KUKA KRL program: EPS_2_25252_SD4A_A_20250910061723.src

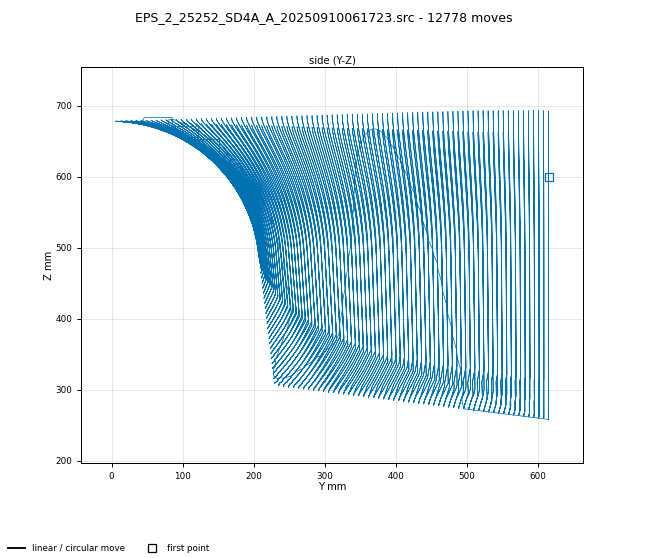
[picture p0: tool path of EPS_2_25252_SD4A_A_20250910061723.src, 12778 of 12780 moves have a stored position in this frame; points joined in program order, loops and branches not executed]
&ACCESS RVP
&REL 4
&COMMENT QRS 19112012
&PARAM EDITMASK = *
DEF PART()
EXT BAS (BAS_COMMAND :IN,REAL :IN )
INT I
BAS (#INITMOV,0 )

;KUKA QRS Post kuka4.cps  Date:22-06-2017 !

File_ID=2837

QRS_PRE_INIT()

;Init var - Until changes are made in qrs_pre_init
Outlet_Square_prg=0
Inlet_1_Square_prg=0
Inlet_2_Square_prg=0
Inlet_3_Square_prg=0
Inlet_4_Square_prg=0
Inlet_5_Square_prg=0

Outlet_1={X 0.000, Y 512.630, Z 510.000, B 0.000, E1 0.000 }
Inlet_1={X 0.000, Y 514.870, Z 480.000, B 0.000, E1 180.000 }
Outlet_1_type=366
Inlet_1_type=366
;QRS#1=Sidecore dimensions
;QRS#2=375-15" PVC SDR 35
;QRS#3=375-15" PVC SDR 35
;QRS#4=
;QRS#5=
;QRS#6=
;QRS#7=
;QRS#8=
;QRS#9=20Y PSX
;QRS#10=20Y PSX
;QRS#11=
;QRS#12=
;QRS#13=
;QRS#14=
;QRS#15=
;QRS#16=1220x127x991 3,25'
;QRS#17=EPS Height
;QRS#18=693
;QRS#19=*
;QRS#20= UPDATED VERSION 22-06-2017
;QRS#21=*
Outlet_Square=0250
Inlet_1_Square=0250
Inlet_2_Square=0
Inlet_3_Square=0
Inlet_4_Square=0
Inlet_5_Square=0
Mill_Square=1
Outlet_Square_Prg=252
Inlet_1_Square_prg=252

QRS_INIT()

$ADVANCE=5

; T1
PTP {E1 173.613,E2 173.613}
PTP {X 0,Y 615.489,A -85,B 0,C 180,E1 173.613,E2 173.613,E3 0,E4 0,E5 0,E6 0}
QRS_SPEED_INIT()
LIN {X 0,Y 615.489,Z 600,A -85,B 0,C 180,E1 173.613,E2 173.613,E3 0,E4 0,E5 0,E6 0} C_VEL
LIN {X 0,Y 615.489,Z 268.179,A -85,B 0,C 180,E1 173.613,E2 173.613} C_VEL
LIN {X 0,Y 615.489,Z 260.004,A -85,B 0,C 180,E1 173.613,E2 173.613} C_VEL
LIN {X 0,Y 615.477,Z 258.004,A -85,B 0,C 180,E1 173.427,E2 173.427} C_VEL
LIN {X 0,Y 615.484,Z 258.009,A -85,B 0,C 180,E1 170.801,E2 170.801} C_VEL
LIN {X 0,Y 615.489,Z 257.994,A -85,B 0,C 180,E1 168.139,E2 168.139} C_VEL
LIN {X 0,Y 615.478,Z 258.004,A -85,B 0,C 180,E1 165.451,E2 165.451} C_VEL
LIN {X 0,Y 615.479,Z 258.006,A -85,B 0,C 180,E1 162.729,E2 162.729} C_VEL
LIN {X 0,Y 615.488,Z 257.994,A -85,B 0,C 180,E1 159.967,E2 159.967} C_VEL
LIN {X 0,Y 615.485,Z 258.012,A -85,B 0,C 180,E1 157.155,E2 157.155} C_VEL
LIN {X 0,Y 615.476,Z 257.998,A -85,B 0,C 180,E1 154.284,E2 154.284} C_VEL
LIN {X 0,Y 615.481,Z 258.002,A -85,B 0,C 180,E1 151.55,E2 151.55} C_VEL
LIN {X 0,Y 615.478,Z 258.01,A -85,B 0,C 180,E1 148.915,E2 148.915} C_VEL
LIN {X 0,Y 615.493,Z 257.994,A -85,B 0,C 180,E1 145.978,E2 145.978} C_VEL
LIN {X 0,Y 615.483,Z 258.014,A -85,B 0,C 180,E1 143.063,E2 143.063} C_VEL
LIN {X 0,Y 615.476,Z 257.997,A -85,B 0,C 180,E1 140.249,E2 140.249} C_VEL
LIN {X 0,Y 615.484,Z 258.001,A -85,B 0,C 180,E1 137.647,E2 137.647} C_VEL
LIN {X 0,Y 615.479,Z 258.008,A -85,B 0,C 180,E1 134.931,E2 134.931} C_VEL
LIN {X 0,Y 615.488,Z 257.994,A -85,B 0,C 180,E1 132.08,E2 132.08} C_VEL
LIN {X 0,Y 615.486,Z 258.01,A -85,B 0,C 180,E1 129.062,E2 129.062} C_VEL
LIN {X 0,Y 615.469,Z 258,A -85,B 0,C 180,E1 126.426,E2 126.426} C_VEL
LIN {X 0,Y 615.487,Z 258.005,A -85,B 0,C 180,E1 123.534,E2 123.534} C_VEL
LIN {X 0,Y 615.47,Z 258.008,A -85,B 0,C 180,E1 120.92,E2 120.92} C_VEL
LIN {X 0,Y 615.467,Z 258,A -85,B 0,C 180,E1 118.447,E2 118.447} C_VEL
LIN {X 0,Y 615.488,Z 258.005,A -85,B 0,C 180,E1 115.569,E2 115.569} C_VEL
LIN {X 0,Y 615.477,Z 258.065,A -85,B 0,C 180,E1 114.239,E2 114.239} C_VEL
LIN {X 0,Y 615.49,Z 282.739,A -85,B 0,C 180,E1 111.982,E2 111.982} C_VEL
LIN {X 0,Y 615.49,Z 489.333,A -85,B 0,C 180,E1 109.424,E2 109.424} C_VEL
LIN {X 0,Y 615.49,Z 505.929,A -85,B 0,C 180,E1 109.078,E2 109.078} C_VEL
LIN {X 0,Y 615.495,Z 522.043,A -85,B 0,C 180,E1 108.607,E2 108.607} C_VEL
LIN {X 0,Y 615.494,Z 537.183,A -85,B 0,C 180,E1 108.038,E2 108.038} C_VEL
LIN {X 0,Y 615.496,Z 551.837,A -85,B 0,C 180,E1 107.356,E2 107.356} C_VEL
LIN {X 0,Y 615.497,Z 566.761,A -85,B 0,C 180,E1 106.51,E2 106.51} C_VEL
LIN {X 0,Y 615.496,Z 580.745,A -85,B 0,C 180,E1 105.565,E2 105.565} C_VEL
LIN {X 0,Y 615.497,Z 593.514,A -85,B 0,C 180,E1 104.549,E2 104.549} C_VEL
LIN {X 0,Y 615.498,Z 604.488,A -85,B 0,C 180,E1 103.537,E2 103.537} C_VEL
LIN {X 0,Y 615.488,Z 615.378,A -85,B 0,C 180,E1 102.363,E2 102.363} C_VEL
LIN {X 0,Y 615.487,Z 625.791,A -85,B 0,C 180,E1 101.041,E2 101.041} C_VEL
LIN {X 0,Y 615.495,Z 634.704,A -85,B 0,C 180,E1 99.696,E2 99.696} C_VEL
LIN {X 0,Y 615.488,Z 641.269,A -85,B 0,C 180,E1 98.537,E2 98.537} C_VEL
LIN {X 0,Y 615.494,Z 648.799,A -85,B 0,C 180,E1 96.897,E2 96.897} C_VEL
LIN {X 0,Y 615.495,Z 654.596,A -85,B 0,C 180,E1 95.241,E2 95.241} C_VEL
LIN {X 0,Y 615.496,Z 657.978,A -85,B 0,C 180,E1 93.928,E2 93.928} C_VEL
LIN {X 0,Y 615.486,Z 660.43,A -85,B 0,C 180,E1 92.618,E2 92.618} C_VEL
LIN {X 0,Y 615.489,Z 661.838,A -85,B 0,C 180,E1 91.309,E2 91.309} C_VEL
LIN {X 0,Y 615.491,Z 662.385,A -85,B 0,C 180,E1 90,E2 90} C_VEL
LIN {X 0,Y 615.486,Z 661.902,A -85,B 0,C 180,E1 88.691,E2 88.691} C_VEL
LIN {X 0,Y 615.486,Z 660.57,A -85,B 0,C 180,E1 87.382,E2 87.382} C_VEL
LIN {X 0,Y 615.493,Z 658.174,A -85,B 0,C 180,E1 86.072,E2 86.072} C_VEL
LIN {X 0,Y 615.49,Z 654.879,A -85,B 0,C 180,E1 84.759,E2 84.759} C_VEL
LIN {X 0,Y 615.491,Z 649.16,A -85,B 0,C 180,E1 83.103,E2 83.103} C_VEL
LIN {X 0,Y 615.497,Z 643.327,A -85,B 0,C 180,E1 81.794,E2 81.794} C_VEL
LIN {X 0,Y 615.492,Z 635.251,A -85,B 0,C 180,E1 80.304,E2 80.304} C_VEL
LIN {X 0,Y 615.493,Z 626.455,A -85,B 0,C 180,E1 78.959,E2 78.959} C_VEL
LIN {X 0,Y 615.491,Z 616.172,A -85,B 0,C 180,E1 77.638,E2 77.638} C_VEL
LIN {X 0,Y 615.495,Z 605.357,A -85,B 0,C 180,E1 76.463,E2 76.463} C_VEL
LIN {X 0,Y 615.495,Z 594.546,A -85,B 0,C 180,E1 75.451,E2 75.451} C_VEL
LIN {X 0,Y 615.497,Z 580.815,A -85,B 0,C 180,E1 74.35,E2 74.35} C_VEL
LIN {X 0,Y 615.498,Z 566.994,A -85,B 0,C 180,E1 73.414,E2 73.414} C_VEL
LIN {X 0,Y 615.492,Z 551.926,A -85,B 0,C 180,E1 72.558,E2 72.558} C_VEL
LIN {X 0,Y 615.487,Z 535.522,A -85,B 0,C 180,E1 71.8,E2 71.8} C_VEL
LIN {X 0,Y 615.489,Z 519.7,A -85,B 0,C 180,E1 71.225,E2 71.225} C_VEL
LIN {X 0,Y 615.497,Z 504.25,A -85,B 0,C 180,E1 70.793,E2 70.793} C_VEL
LIN {X 0,Y 615.488,Z 488.065,A -85,B 0,C 180,E1 70.467,E2 70.467} C_VEL
LIN {X 0,Y 615.489,Z 282.76,A -85,B 0,C 180,E1 67.93,E2 67.93} C_VEL
LIN {X 0,Y 615.467,Z 257.999,A -85,B 0,C 180,E1 65.66,E2 65.66} C_VEL
LIN {X 0,Y 615.468,Z 258.009,A -85,B 0,C 180,E1 62.959,E2 62.959} C_VEL
LIN {X 0,Y 615.491,Z 258,A -85,B 0,C 180,E1 60.205,E2 60.205} C_VEL
LIN {X 0,Y 615.462,Z 258.001,A -85,B 0,C 180,E1 57.541,E2 57.541} C_VEL
LIN {X 0,Y 615.463,Z 258.006,A -85,B 0,C 180,E1 55.184,E2 55.184} C_VEL
LIN {X 0,Y 615.487,Z 258.014,A -85,B 0,C 180,E1 52.758,E2 52.758} C_VEL
LIN {X 0,Y 615.49,Z 257.995,A -85,B 0,C 180,E1 49.911,E2 49.911} C_VEL
LIN {X 0,Y 615.47,Z 257.999,A -85,B 0,C 180,E1 47.646,E2 47.646} C_VEL
LIN {X 0,Y 615.476,Z 258.011,A -85,B 0,C 180,E1 44.931,E2 44.931} C_VEL
LIN {X 0,Y 615.492,Z 257.996,A -85,B 0,C 180,E1 42.081,E2 42.081} C_VEL
LIN {X 0,Y 615.477,Z 257.997,A -85,B 0,C 180,E1 39.751,E2 39.751} C_VEL
LIN {X 0,Y 615.479,Z 258.012,A -85,B 0,C 180,E1 36.936,E2 36.936} C_VEL
LIN {X 0,Y 615.491,Z 257.995,A -85,B 0,C 180,E1 34.022,E2 34.022} C_VEL
LIN {X 0,Y 615.475,Z 257.998,A -85,B 0,C 180,E1 31.686,E2 31.686} C_VEL
LIN {X 0,Y 615.469,Z 258.003,A -85,B 0,C 180,E1 29.407,E2 29.407} C_VEL
LIN {X 0,Y 615.483,Z 258.009,A -85,B 0,C 180,E1 27.045,E2 27.045} C_VEL
LIN {X 0,Y 615.485,Z 257.999,A -85,B 0,C 180,E1 24.272,E2 24.272} C_VEL
LIN {X 0,Y 615.471,Z 258.002,A -85,B 0,C 180,E1 21.433,E2 21.433} C_VEL
LIN {X 0,Y 615.484,Z 258.006,A -85,B 0,C 180,E1 18.605,E2 18.605} C_VEL
LIN {X 0,Y 615.486,Z 257.995,A -85,B 0,C 180,E1 15.905,E2 15.905} C_VEL
LIN {X 0,Y 615.478,Z 258.008,A -85,B 0,C 180,E1 13.201,E2 13.201} C_VEL
LIN {X 0,Y 615.48,Z 258.003,A -85,B 0,C 180,E1 10.527,E2 10.527} C_VEL
LIN {X 0,Y 615.487,Z 257.995,A -85,B 0,C 180,E1 7.876,E2 7.876} C_VEL
LIN {X 0,Y 615.481,Z 258.007,A -85,B 0,C 180,E1 5.241,E2 5.241} C_VEL
LIN {X 0,Y 615.479,Z 258.005,A -85,B 0,C 180,E1 2.618,E2 2.618} C_VEL
LIN {X 0,Y 615.486,Z 257.995,A -85,B 0,C 180,E1 0,E2 0} C_VEL
LIN {X 0,Y 615.479,Z 258.005,A -85,B 0,C 180,E1 -2.618,E2 -2.618} C_VEL
LIN {X 0,Y 615.481,Z 258.007,A -85,B 0,C 180,E1 -5.241,E2 -5.241} C_VEL
LIN {X 0,Y 615.487,Z 257.995,A -85,B 0,C 180,E1 -7.876,E2 -7.876} C_VEL
LIN {X 0,Y 615.48,Z 258.003,A -85,B 0,C 180,E1 -10.527,E2 -10.527} C_VEL
LIN {X 0,Y 615.478,Z 258.008,A -85,B 0,C 180,E1 -13.201,E2 -13.201} C_VEL
LIN {X 0,Y 615.486,Z 257.995,A -85,B 0,C 180,E1 -15.905,E2 -15.905} C_VEL
LIN {X 0,Y 615.485,Z 258.007,A -85,B 0,C 180,E1 -18.646,E2 -18.646} C_VEL
LIN {X 0,Y 615.471,Z 258.002,A -85,B 0,C 180,E1 -21.432,E2 -21.432} C_VEL
LIN {X 0,Y 615.485,Z 257.999,A -85,B 0,C 180,E1 -24.272,E2 -24.272} C_VEL
LIN {X 0,Y 615.475,Z 258.007,A -85,B 0,C 180,E1 -27.178,E2 -27.178} C_VEL
LIN {X 0,Y 615.482,Z 257.996,A -85,B 0,C 180,E1 -29.795,E2 -29.795} C_VEL
LIN {X 0,Y 615.485,Z 258.004,A -85,B 0,C 180,E1 -32.457,E2 -32.457} C_VEL
LIN {X 0,Y 615.498,Z 258.013,A -85,B 0,C 180,E1 -34.814,E2 -34.814} C_VEL
LIN {X 0,Y 615.469,Z 258.005,A -85,B 0,C 180,E1 -37.243,E2 -37.243} C_VEL
LIN {X 0,Y 615.494,Z 257.995,A -85,B 0,C 180,E1 -40.09,E2 -40.09} C_VEL
LIN {X 0,Y 615.475,Z 258.008,A -85,B 0,C 180,E1 -43.047,E2 -43.047} C_VEL
LIN {X 0,Y 615.485,Z 257.995,A -85,B 0,C 180,E1 -45.851,E2 -45.851} C_VEL
LIN {X 0,Y 615.49,Z 258.007,A -85,B 0,C 180,E1 -48.527,E2 -48.527} C_VEL
LIN {X 0,Y 615.468,Z 258.007,A -85,B 0,C 180,E1 -51.095,E2 -51.095} C_VEL
LIN {X 0,Y 615.466,Z 258,A -85,B 0,C 180,E1 -53.574,E2 -53.574} C_VEL
LIN {X 0,Y 615.49,Z 258.007,A -85,B 0,C 180,E1 -56.465,E2 -56.465} C_VEL
LIN {X 0,Y 615.466,Z 258.007,A -85,B 0,C 180,E1 -59.079,E2 -59.079} C_VEL
LIN {X 0,Y 615.463,Z 258,A -85,B 0,C 180,E1 -61.553,E2 -61.553} C_VEL
LIN {X 0,Y 615.465,Z 258.187,A -85,B 0,C 180,E1 -63.601,E2 -63.601} C_VEL
LIN {X 0,Y 615.476,Z 290.169,A -85,B 0,C 180,E1 -66.217,E2 -66.217} C_VEL
LIN {X 0,Y 615.493,Z 312.014,A -85,B 0,C 180,E1 -67.974,E2 -67.974} C_VEL
LIN {X 0,Y 615.491,Z 519.442,A -85,B 0,C 180,E1 -70.532,E2 -70.532} C_VEL
LIN {X 0,Y 615.493,Z 536.004,A -85,B 0,C 180,E1 -70.879,E2 -70.879} C_VEL
LIN {X 0,Y 615.493,Z 550.938,A -85,B 0,C 180,E1 -71.311,E2 -71.311} C_VEL
LIN {X 0,Y 615.491,Z 566.351,A -85,B 0,C 180,E1 -71.881,E2 -71.881} C_VEL
LIN {X 0,Y 615.493,Z 581.008,A -85,B 0,C 180,E1 -72.558,E2 -72.558} C_VEL
LIN {X 0,Y 615.5,Z 594.839,A -85,B 0,C 180,E1 -73.329,E2 -73.329} C_VEL
LIN {X 0,Y 615.499,Z 609.04,A -85,B 0,C 180,E1 -74.265,E2 -74.265} C_VEL
LIN {X 0,Y 615.495,Z 622.094,A -85,B 0,C 180,E1 -75.282,E2 -75.282} C_VEL
LIN {X 0,Y 615.494,Z 633.215,A -85,B 0,C 180,E1 -76.295,E2 -76.295} C_VEL
LIN {X 0,Y 615.493,Z 644.292,A -85,B 0,C 180,E1 -77.47,E2 -77.47} C_VEL
LIN {X 0,Y 615.494,Z 653.767,A -85,B 0,C 180,E1 -78.64,E2 -78.64} C_VEL
LIN {X 0,Y 615.496,Z 662.965,A -85,B 0,C 180,E1 -79.972,E2 -79.972} C_VEL
LIN {X 0,Y 615.489,Z 671.502,A -85,B 0,C 180,E1 -81.463,E2 -81.463} C_VEL
LIN {X 0,Y 615.491,Z 678.982,A -85,B 0,C 180,E1 -83.102,E2 -83.102} C_VEL
LIN {X 0,Y 615.492,Z 684.741,A -85,B 0,C 180,E1 -84.759,E2 -84.759} C_VEL
LIN {X 0,Y 615.494,Z 688.076,A -85,B 0,C 180,E1 -86.072,E2 -86.072} C_VEL
LIN {X 0,Y 615.485,Z 690.504,A -85,B 0,C 180,E1 -87.382,E2 -87.382} C_VEL
LIN {X 0,Y 615.488,Z 691.87,A -85,B 0,C 180,E1 -88.691,E2 -88.691} C_VEL
LIN {X 0,Y 615.489,Z 692.39,A -85,B 0,C 180,E1 -90,E2 -90} C_VEL
LIN {X 0,Y 615.488,Z 691.87,A -85,B 0,C 180,E1 -91.309,E2 -91.309} C_VEL
LIN {X 0,Y 615.485,Z 690.504,A -85,B 0,C 180,E1 -92.618,E2 -92.618} C_VEL
LIN {X 0,Y 615.494,Z 688.076,A -85,B 0,C 180,E1 -93.928,E2 -93.928} C_VEL
LIN {X 0,Y 615.492,Z 684.741,A -85,B 0,C 180,E1 -95.241,E2 -95.241} C_VEL
LIN {X 0,Y 615.491,Z 678.982,A -85,B 0,C 180,E1 -96.898,E2 -96.898} C_VEL
LIN {X 0,Y 615.489,Z 671.502,A -85,B 0,C 180,E1 -98.537,E2 -98.537} C_VEL
LIN {X 0,Y 615.496,Z 662.964,A -85,B 0,C 180,E1 -100.028,E2 -100.028} C_VEL
LIN {X 0,Y 615.494,Z 653.767,A -85,B 0,C 180,E1 -101.36,E2 -101.36} C_VEL
LIN {X 0,Y 615.495,Z 644.291,A -85,B 0,C 180,E1 -102.53,E2 -102.53} C_VEL
LIN {X 0,Y 615.494,Z 633.214,A -85,B 0,C 180,E1 -103.706,E2 -103.706} C_VEL
LIN {X 0,Y 615.495,Z 621.116,A -85,B 0,C 180,E1 -104.802,E2 -104.802} C_VEL
LIN {X 0,Y 615.498,Z 606.71,A -85,B 0,C 180,E1 -105.905,E2 -105.905} C_VEL
LIN {X 0,Y 615.497,Z 592.016,A -85,B 0,C 180,E1 -106.842,E2 -106.842} C_VEL
LIN {X 0,Y 615.49,Z 577.512,A -85,B 0,C 180,E1 -107.613,E2 -107.613} C_VEL
LIN {X 0,Y 615.49,Z 562.248,A -85,B 0,C 180,E1 -108.282,E2 -108.282} C_VEL
LIN {X 0,Y 615.49,Z 546.997,A -85,B 0,C 180,E1 -108.818,E2 -108.818} C_VEL
LIN {X 0,Y 615.497,Z 530.524,A -85,B 0,C 180,E1 -109.251,E2 -109.251} C_VEL
LIN {X 0,Y 615.49,Z 514.936,A -85,B 0,C 180,E1 -109.533,E2 -109.533} C_VEL
LIN {X 0,Y 615.492,Z 312.014,A -85,B 0,C 180,E1 -112.026,E2 -112.026} C_VEL
LIN {X 0,Y 615.458,Z 276.405,A -85,B 0,C 180,E1 -114.903,E2 -114.903} C_VEL
LIN {X 0,Y 615.464,Z 258,A -85,B 0,C 180,E1 -116.422,E2 -116.422} C_VEL
LIN {X 0,Y 615.458,Z 258.003,A -85,B 0,C 180,E1 -118.659,E2 -118.659} C_VEL
LIN {X 0,Y 615.476,Z 258.009,A -85,B 0,C 180,E1 -121.084,E2 -121.084} C_VEL
LIN {X 0,Y 615.492,Z 257.995,A -85,B 0,C 180,E1 -124.021,E2 -124.021} C_VEL
LIN {X 0,Y 615.465,Z 258,A -85,B 0,C 180,E1 -126.426,E2 -126.426} C_VEL
LIN {X 0,Y 615.475,Z 258.01,A -85,B 0,C 180,E1 -129.061,E2 -129.061} C_VEL
LIN {X 0,Y 615.491,Z 258.007,A -85,B 0,C 180,E1 -131.473,E2 -131.473} C_VEL
LIN {X 0,Y 615.485,Z 257.995,A -85,B 0,C 180,E1 -134.149,E2 -134.149} C_VEL
LIN {X 0,Y 615.474,Z 258.008,A -85,B 0,C 180,E1 -136.954,E2 -136.954} C_VEL
LIN {X 0,Y 615.494,Z 257.995,A -85,B 0,C 180,E1 -139.91,E2 -139.91} C_VEL
LIN {X 0,Y 615.467,Z 258.005,A -85,B 0,C 180,E1 -142.757,E2 -142.757} C_VEL
LIN {X 0,Y 615.492,Z 258.011,A -85,B 0,C 180,E1 -145.298,E2 -145.298} C_VEL
LIN {X 0,Y 615.474,Z 257.998,A -85,B 0,C 180,E1 -148.314,E2 -148.314} C_VEL
LIN {X 0,Y 615.467,Z 258.003,A -85,B 0,C 180,E1 -150.593,E2 -150.593} C_VEL
LIN {X 0,Y 615.481,Z 258.009,A -85,B 0,C 180,E1 -152.955,E2 -152.955} C_VEL
LIN {X 0,Y 615.485,Z 257.999,A -85,B 0,C 180,E1 -155.728,E2 -155.728} C_VEL
LIN {X 0,Y 615.47,Z 258.002,A -85,B 0,C 180,E1 -158.568,E2 -158.568} C_VEL
LIN {X 0,Y 615.484,Z 258.007,A -85,B 0,C 180,E1 -161.395,E2 -161.395} C_VEL
LIN {X 0,Y 615.486,Z 257.995,A -85,B 0,C 180,E1 -164.095,E2 -164.095} C_VEL
LIN {X 0,Y 615.477,Z 258.007,A -85,B 0,C 180,E1 -166.799,E2 -166.799} C_VEL
LIN {X 0,Y 615.482,Z 258.004,A -85,B 0,C 180,E1 -169.473,E2 -169.473} C_VEL
LIN {X 0,Y 615.487,Z 257.995,A -85,B 0,C 180,E1 -172.124,E2 -172.124} C_VEL
LIN {X 0,Y 615.478,Z 258.007,A -85,B 0,C 180,E1 -174.759,E2 -174.759} C_VEL
LIN {X 0,Y 615.481,Z 258.005,A -85,B 0,C 180,E1 -177.382,E2 -177.382} C_VEL
LIN {X 0,Y 615.486,Z 257.995,A -85,B 0,C 180,E1 -180,E2 -180} C_VEL
LIN {X 0,Y 615.476,Z 258.004,A -85,B 0,C 180,E1 -182.618,E2 -182.618} C_VEL
LIN {X 0,Y 615.483,Z 258.008,A -85,B 0,C 180,E1 -185.241,E2 -185.241} C_VEL
LIN {X 0,Y 615.477,Z 258.004,A -85,B 0,C 180,E1 -186.573,E2 -186.573} C_VEL
LIN {X 0,Y 614.806,Z 258.156,A -85,B 0,C 180,E1 -187.119,E2 -187.119} C_VEL
LIN {X 0,Y 611.975,Z 258.561,A -85,B 0,C 180,E1 -188.005,E2 -188.005} C_VEL
LIN {X 0,Y 609.583,Z 258.875,A -85,B 0,C 180,E1 -188.718,E2 -188.718} C_VEL
LIN {X 0,Y 608.548,Z 258.994,A -85,B 0,C 180,E1 -189.267,E2 -189.267} C_VEL
LIN {X 0,Y 608.458,Z 259.002,A -85,B 0,C 180,E1 -189.454,E2 -189.454} C_VEL
LIN {X 0,Y 608.462,Z 258.998,A -85,B 0,C 180,E1 -192,E2 -192} C_VEL
LIN {X 0,Y 608.469,Z 259.004,A -85,B 0,C 180,E1 -194.721,E2 -194.721} C_VEL
LIN {X 0,Y 608.45,Z 259.003,A -85,B 0,C 180,E1 -197.477,E2 -197.477} C_VEL
LIN {X 0,Y 608.46,Z 259,A -85,B 0,C 180,E1 -200.274,E2 -200.274} C_VEL
LIN {X 0,Y 608.446,Z 259.008,A -85,B 0,C 180,E1 -203.124,E2 -203.124} C_VEL
LIN {X 0,Y 608.462,Z 258.999,A -85,B 0,C 180,E1 -205.72,E2 -205.72} C_VEL
LIN {X 0,Y 608.448,Z 259.001,A -85,B 0,C 180,E1 -208.267,E2 -208.267} C_VEL
LIN {X 0,Y 608.474,Z 259.002,A -85,B 0,C 180,E1 -210.545,E2 -210.545} C_VEL
LIN {X 0,Y 608.451,Z 259.011,A -85,B 0,C 180,E1 -212.88,E2 -212.88} C_VEL
LIN {X 0,Y 608.439,Z 259.005,A -85,B 0,C 180,E1 -215.278,E2 -215.278} C_VEL
LIN {X 0,Y 608.465,Z 258.998,A -85,B 0,C 180,E1 -217.747,E2 -217.747} C_VEL
LIN {X 0,Y 608.455,Z 259.002,A -85,B 0,C 180,E1 -220.33,E2 -220.33} C_VEL
LIN {X 0,Y 608.449,Z 259.009,A -85,B 0,C 180,E1 -222.96,E2 -222.96} C_VEL
LIN {X 0,Y 608.455,Z 258.999,A -85,B 0,C 180,E1 -225.736,E2 -225.736} C_VEL
LIN {X 0,Y 608.461,Z 259.007,A -85,B 0,C 180,E1 -228.658,E2 -228.658} C_VEL
LIN {X 0,Y 608.462,Z 259,A -85,B 0,C 180,E1 -231.412,E2 -231.412} C_VEL
LIN {X 0,Y 608.446,Z 259.001,A -85,B 0,C 180,E1 -233.955,E2 -233.955} C_VEL
LIN {X 0,Y 608.466,Z 259.002,A -85,B 0,C 180,E1 -236.33,E2 -236.33} C_VEL
LIN {X 0,Y 608.46,Z 259.009,A -85,B 0,C 180,E1 -238.73,E2 -238.73} C_VEL
LIN {X 0,Y 608.456,Z 259.001,A -85,B 0,C 180,E1 -241.383,E2 -241.383} C_VEL
LIN {X 0,Y 608.438,Z 259.002,A -85,B 0,C 180,E1 -243.964,E2 -243.964} C_VEL
LIN {X 0,Y 608.464,Z 259.047,A -85,B 0,C 180,E1 -245.554,E2 -245.554} C_VEL
LIN {X 0,Y 608.742,Z 263.037,A -85,B 0,C 180,E1 -245.938,E2 -245.938} C_VEL
LIN {X 0,Y 608.741,Z 283.15,A -85,B 0,C 180,E1 -247.778,E2 -247.778} C_VEL
LIN {X 0,Y 608.876,Z 337.239,A -85,B 0,C 180,E1 -248.457,E2 -248.457} C_VEL
LIN {X 0,Y 608.802,Z 489.369,A -85,B 0,C 180,E1 -250.354,E2 -250.354} C_VEL
LIN {X 0,Y 608.775,Z 505.041,A -85,B 0,C 180,E1 -250.681,E2 -250.681} C_VEL
LIN {X 0,Y 608.743,Z 520.901,A -85,B 0,C 180,E1 -251.14,E2 -251.14} C_VEL
LIN {X 0,Y 608.7,Z 535.318,A -85,B 0,C 180,E1 -251.672,E2 -251.672} C_VEL
LIN {X 0,Y 608.681,Z 551.851,A -85,B 0,C 180,E1 -252.444,E2 -252.444} C_VEL
LIN {X 0,Y 608.619,Z 565.517,A -85,B 0,C 180,E1 -253.221,E2 -253.221} C_VEL
LIN {X 0,Y 608.592,Z 579.601,A -85,B 0,C 180,E1 -254.168,E2 -254.168} C_VEL
LIN {X 0,Y 608.557,Z 591.616,A -85,B 0,C 180,E1 -255.111,E2 -255.111} C_VEL
LIN {X 0,Y 608.515,Z 604.574,A -85,B 0,C 180,E1 -256.305,E2 -256.305} C_VEL
LIN {X 0,Y 608.489,Z 615.516,A -85,B 0,C 180,E1 -257.493,E2 -257.493} C_VEL
LIN {X 0,Y 608.458,Z 624.877,A -85,B 0,C 180,E1 -258.676,E2 -258.676} C_VEL
LIN {X 0,Y 608.471,Z 633.987,A -85,B 0,C 180,E1 -260.023,E2 -260.023} C_VEL
LIN {X 0,Y 608.444,Z 641.618,A -85,B 0,C 180,E1 -261.364,E2 -261.364} C_VEL
LIN {X 0,Y 608.439,Z 647.857,A -85,B 0,C 180,E1 -262.7,E2 -262.7} C_VEL
LIN {X 0,Y 608.432,Z 652.98,A -85,B 0,C 180,E1 -264.033,E2 -264.033} C_VEL
LIN {X 0,Y 608.429,Z 656.935,A -85,B 0,C 180,E1 -265.362,E2 -265.362} C_VEL
LIN {X 0,Y 608.416,Z 659.907,A -85,B 0,C 180,E1 -266.689,E2 -266.689} C_VEL
LIN {X 0,Y 608.442,Z 661.835,A -85,B 0,C 180,E1 -268.014,E2 -268.014} C_VEL
LIN {X 0,Y 608.434,Z 662.84,A -85,B 0,C 180,E1 -269.338,E2 -269.338} C_VEL
LIN {X 0,Y 608.434,Z 662.861,A -85,B 0,C 180,E1 -270.662,E2 -270.662} C_VEL
LIN {X 0,Y 608.443,Z 661.942,A -85,B 0,C 180,E1 -271.986,E2 -271.986} C_VEL
LIN {X 0,Y 608.419,Z 660.057,A -85,B 0,C 180,E1 -273.311,E2 -273.311} C_VEL
LIN {X 0,Y 608.425,Z 657.176,A -85,B 0,C 180,E1 -274.638,E2 -274.638} C_VEL
LIN {X 0,Y 608.433,Z 653.267,A -85,B 0,C 180,E1 -275.967,E2 -275.967} C_VEL
LIN {X 0,Y 608.438,Z 648.242,A -85,B 0,C 180,E1 -277.3,E2 -277.3} C_VEL
LIN {X 0,Y 608.444,Z 642.085,A -85,B 0,C 180,E1 -278.636,E2 -278.636} C_VEL
LIN {X 0,Y 608.461,Z 633.517,A -85,B 0,C 180,E1 -280.145,E2 -280.145} C_VEL
LIN {X 0,Y 608.466,Z 624.299,A -85,B 0,C 180,E1 -281.493,E2 -281.493} C_VEL
LIN {X 0,Y 608.496,Z 613.328,A -85,B 0,C 180,E1 -282.846,E2 -282.846} C_VEL
LIN {X 0,Y 608.52,Z 601.976,A -85,B 0,C 180,E1 -284.036,E2 -284.036} C_VEL
LIN {X 0,Y 608.548,Z 589.588,A -85,B 0,C 180,E1 -285.147,E2 -285.147} C_VEL
LIN {X 0,Y 608.607,Z 577.33,A -85,B 0,C 180,E1 -286.09,E2 -286.09} C_VEL
LIN {X 0,Y 608.622,Z 562.754,A -85,B 0,C 180,E1 -287.038,E2 -287.038} C_VEL
LIN {X 0,Y 608.657,Z 548.423,A -85,B 0,C 180,E1 -287.817,E2 -287.817} C_VEL
LIN {X 0,Y 608.716,Z 533.427,A -85,B 0,C 180,E1 -288.492,E2 -288.492} C_VEL
LIN {X 0,Y 608.755,Z 517.043,A -85,B 0,C 180,E1 -289.078,E2 -289.078} C_VEL
LIN {X 0,Y 608.778,Z 500.575,A -85,B 0,C 180,E1 -289.516,E2 -289.516} C_VEL
LIN {X 0,Y 608.795,Z 485.014,A -85,B 0,C 180,E1 -289.8,E2 -289.8} C_VEL
LIN {X 0,Y 608.822,Z 283.654,A -85,B 0,C 180,E1 -292.302,E2 -292.302} C_VEL
LIN {X 0,Y 608.668,Z 282.51,A -85,B 0,C 180,E1 -292.353,E2 -292.353} C_VEL
LIN {X 0,Y 608.653,Z 260.012,A -85,B 0,C 180,E1 -294.438,E2 -294.438} C_VEL
LIN {X 0,Y 608.43,Z 259.005,A -85,B 0,C 180,E1 -294.572,E2 -294.572} C_VEL
LIN {X 0,Y 608.469,Z 259.006,A -85,B 0,C 180,E1 -297.206,E2 -297.206} C_VEL
LIN {X 0,Y 608.469,Z 258.999,A -85,B 0,C 180,E1 -299.972,E2 -299.972} C_VEL
LIN {X 0,Y 608.449,Z 259.004,A -85,B 0,C 180,E1 -302.88,E2 -302.88} C_VEL
LIN {X 0,Y 608.436,Z 259.013,A -85,B 0,C 180,E1 -305.278,E2 -305.278} C_VEL
LIN {X 0,Y 608.469,Z 259.001,A -85,B 0,C 180,E1 -307.746,E2 -307.746} C_VEL
LIN {X 0,Y 608.443,Z 259.001,A -85,B 0,C 180,E1 -310.328,E2 -310.328} C_VEL
LIN {X 0,Y 608.445,Z 259.006,A -85,B 0,C 180,E1 -312.96,E2 -312.96} C_VEL
LIN {X 0,Y 608.459,Z 259.002,A -85,B 0,C 180,E1 -315.735,E2 -315.735} C_VEL
LIN {X 0,Y 608.446,Z 259.002,A -85,B 0,C 180,E1 -318.659,E2 -318.659} C_VEL
LIN {X 0,Y 608.467,Z 259.005,A -85,B 0,C 180,E1 -321.412,E2 -321.412} C_VEL
LIN {X 0,Y 608.475,Z 258.997,A -85,B 0,C 180,E1 -323.95,E2 -323.95} C_VEL
LIN {X 0,Y 608.443,Z 259.001,A -85,B 0,C 180,E1 -326.328,E2 -326.328} C_VEL
LIN {X 0,Y 608.443,Z 259.004,A -85,B 0,C 180,E1 -328.732,E2 -328.732} C_VEL
LIN {X 0,Y 608.472,Z 259.004,A -85,B 0,C 180,E1 -331.379,E2 -331.379} C_VEL
LIN {X 0,Y 608.462,Z 258.999,A -85,B 0,C 180,E1 -334.28,E2 -334.28} C_VEL
LIN {X 0,Y 608.445,Z 259.007,A -85,B 0,C 180,E1 -336.876,E2 -336.876} C_VEL
LIN {X 0,Y 608.461,Z 259,A -85,B 0,C 180,E1 -339.726,E2 -339.726} C_VEL
LIN {X 0,Y 608.447,Z 259.002,A -85,B 0,C 180,E1 -342.523,E2 -342.523} C_VEL
LIN {X 0,Y 608.469,Z 259.005,A -85,B 0,C 180,E1 -345.279,E2 -345.279} C_VEL
LIN {X 0,Y 608.462,Z 258.999,A -85,B 0,C 180,E1 -348,E2 -348} C_VEL
LIN {X 0,Y 608.464,Z 259.003,A -85,B 0,C 180,E1 -350.694,E2 -350.694} C_VEL
LIN {X 0,Y 608.475,Z 259.002,A -85,B 0,C 180,E1 -353.367,E2 -353.367} C_VEL
LIN {X 0,Y 608.456,Z 258.999,A -85,B 0,C 180,E1 -356.026,E2 -356.026} C_VEL
LIN {X 0,Y 608.464,Z 259.003,A -85,B 0,C 180,E1 -358.676,E2 -358.676} C_VEL
LIN {X 0,Y 608.464,Z 259.003,A -85,B 0,C 180,E1 -361.324,E2 -361.324} C_VEL
LIN {X 0,Y 608.456,Z 258.999,A -85,B 0,C 180,E1 -363.974,E2 -363.974} C_VEL
LIN {X 0,Y 608.475,Z 259.002,A -85,B 0,C 180,E1 -366.632,E2 -366.632} C_VEL
LIN {X 0,Y 608.464,Z 259.003,A -85,B 0,C 180,E1 -369.306,E2 -369.306} C_VEL
LIN {X 0,Y 608.462,Z 258.998,A -85,B 0,C 180,E1 -372,E2 -372} C_VEL
LIN {X 0,Y 608.469,Z 259.005,A -85,B 0,C 180,E1 -374.721,E2 -374.721} C_VEL
LIN {X 0,Y 608.447,Z 259.002,A -85,B 0,C 180,E1 -377.477,E2 -377.477} C_VEL
LIN {X 0,Y 608.462,Z 259,A -85,B 0,C 180,E1 -380.274,E2 -380.274} C_VEL
LIN {X 0,Y 608.445,Z 259.007,A -85,B 0,C 180,E1 -383.124,E2 -383.124} C_VEL
LIN {X 0,Y 608.46,Z 258.999,A -85,B 0,C 180,E1 -385.72,E2 -385.72} C_VEL
LIN {X 0,Y 608.472,Z 259.004,A -85,B 0,C 180,E1 -388.621,E2 -388.621} C_VEL
LIN {X 0,Y 608.441,Z 259.004,A -85,B 0,C 180,E1 -391.318,E2 -391.318} C_VEL
LIN {X 0,Y 608.468,Z 258.998,A -85,B 0,C 180,E1 -393.735,E2 -393.735} C_VEL
LIN {X 0,Y 608.474,Z 258.998,A -85,B 0,C 180,E1 -396.09,E2 -396.09} C_VEL
LIN {X 0,Y 608.468,Z 259.005,A -85,B 0,C 180,E1 -398.588,E2 -398.588} C_VEL
LIN {X 0,Y 608.446,Z 259.003,A -85,B 0,C 180,E1 -401.341,E2 -401.341} C_VEL
LIN {X 0,Y 608.459,Z 259.002,A -85,B 0,C 180,E1 -404.265,E2 -404.265} C_VEL
LIN {X 0,Y 608.445,Z 259.006,A -85,B 0,C 180,E1 -407.04,E2 -407.04} C_VEL
LIN {X 0,Y 608.449,Z 259,A -85,B 0,C 180,E1 -409.697,E2 -409.697} C_VEL
LIN {X 0,Y 608.467,Z 259.001,A -85,B 0,C 180,E1 -412.254,E2 -412.254} C_VEL
LIN {X 0,Y 608.432,Z 259.006,A -85,B 0,C 180,E1 -415.097,E2 -415.097} C_VEL
LIN {X 0,Y 608.442,Z 259.001,A -85,B 0,C 180,E1 -417.48,E2 -417.48} C_VEL
LIN {X 0,Y 608.475,Z 259.001,A -85,B 0,C 180,E1 -420.221,E2 -420.221} C_VEL
LIN {X 0,Y 608.431,Z 259.006,A -85,B 0,C 180,E1 -423.225,E2 -423.225} C_VEL
LIN {X 0,Y 608.449,Z 259.015,A -85,B 0,C 180,E1 -423.342,E2 -423.342} C_VEL
LIN {X 0,Y 608.824,Z 262.051,A -85,B 0,C 180,E1 -423.614,E2 -423.614} C_VEL
LIN {X 0,Y 608.729,Z 296.28,A -85,B 0,C 180,E1 -426.437,E2 -426.437} C_VEL
LIN {X 0,Y 608.713,Z 312.014,A -85,B 0,C 180,E1 -427.716,E2 -427.716} C_VEL
LIN {X 0,Y 608.9,Z 322.571,A -85,B 0,C 180,E1 -427.857,E2 -427.857} C_VEL
LIN {X 0,Y 608.795,Z 517.952,A -85,B 0,C 180,E1 -430.287,E2 -430.287} C_VEL
LIN {X 0,Y 608.795,Z 534.179,A -85,B 0,C 180,E1 -430.616,E2 -430.616} C_VEL
LIN {X 0,Y 608.737,Z 549.648,A -85,B 0,C 180,E1 -431.052,E2 -431.052} C_VEL
LIN {X 0,Y 608.711,Z 564.372,A -85,B 0,C 180,E1 -431.589,E2 -431.589} C_VEL
LIN {X 0,Y 608.678,Z 579.265,A -85,B 0,C 180,E1 -432.27,E2 -432.27} C_VEL
LIN {X 0,Y 608.616,Z 594.842,A -85,B 0,C 180,E1 -433.134,E2 -433.134} C_VEL
LIN {X 0,Y 608.579,Z 609.048,A -85,B 0,C 180,E1 -434.082,E2 -434.082} C_VEL
LIN {X 0,Y 608.556,Z 622.129,A -85,B 0,C 180,E1 -435.111,E2 -435.111} C_VEL
LIN {X 0,Y 608.528,Z 634.01,A -85,B 0,C 180,E1 -436.204,E2 -436.204} C_VEL
LIN {X 0,Y 608.49,Z 645.913,A -85,B 0,C 180,E1 -437.493,E2 -437.493} C_VEL
LIN {X 0,Y 608.487,Z 655.207,A -85,B 0,C 180,E1 -438.677,E2 -438.677} C_VEL
LIN {X 0,Y 608.471,Z 664.258,A -85,B 0,C 180,E1 -440.023,E2 -440.023} C_VEL
LIN {X 0,Y 608.444,Z 671.858,A -85,B 0,C 180,E1 -441.364,E2 -441.364} C_VEL
LIN {X 0,Y 608.437,Z 679.469,A -85,B 0,C 180,E1 -443.034,E2 -443.034} C_VEL
LIN {X 0,Y 608.435,Z 685.245,A -85,B 0,C 180,E1 -444.698,E2 -444.698} C_VEL
LIN {X 0,Y 608.431,Z 688.633,A -85,B 0,C 180,E1 -446.026,E2 -446.026} C_VEL
LIN {X 0,Y 608.412,Z 691.086,A -85,B 0,C 180,E1 -447.352,E2 -447.352} C_VEL
LIN {X 0,Y 608.441,Z 692.477,A -85,B 0,C 180,E1 -448.676,E2 -448.676} C_VEL
LIN {X 0,Y 608.429,Z 693,A -85,B 0,C 180,E1 -450,E2 -450} C_VEL
LIN {X 0,Y 608.441,Z 692.477,A -85,B 0,C 180,E1 -451.324,E2 -451.324} C_VEL
LIN {X 0,Y 608.412,Z 691.086,A -85,B 0,C 180,E1 -452.648,E2 -452.648} C_VEL
LIN {X 0,Y 608.431,Z 688.632,A -85,B 0,C 180,E1 -453.974,E2 -453.974} C_VEL
LIN {X 0,Y 608.435,Z 685.245,A -85,B 0,C 180,E1 -455.302,E2 -455.302} C_VEL
LIN {X 0,Y 608.437,Z 679.469,A -85,B 0,C 180,E1 -456.966,E2 -456.966} C_VEL
LIN {X 0,Y 608.444,Z 671.858,A -85,B 0,C 180,E1 -458.636,E2 -458.636} C_VEL
LIN {X 0,Y 608.462,Z 663.245,A -85,B 0,C 180,E1 -460.145,E2 -460.145} C_VEL
LIN {X 0,Y 608.466,Z 653.968,A -85,B 0,C 180,E1 -461.493,E2 -461.493} C_VEL
LIN {X 0,Y 608.49,Z 644.422,A -85,B 0,C 180,E1 -462.677,E2 -462.677} C_VEL
LIN {X 0,Y 608.521,Z 632.965,A -85,B 0,C 180,E1 -463.896,E2 -463.896} C_VEL
LIN {X 0,Y 608.553,Z 621.144,A -85,B 0,C 180,E1 -464.975,E2 -464.975} C_VEL
LIN {X 0,Y 608.607,Z 606.711,A -85,B 0,C 180,E1 -466.09,E2 -466.09} C_VEL
LIN {X 0,Y 608.648,Z 592.019,A -85,B 0,C 180,E1 -467.038,E2 -467.038} C_VEL
LIN {X 0,Y 608.659,Z 577.515,A -85,B 0,C 180,E1 -467.817,E2 -467.817} C_VEL
LIN {X 0,Y 608.718,Z 562.251,A -85,B 0,C 180,E1 -468.493,E2 -468.493} C_VEL
LIN {X 0,Y 608.748,Z 546.244,A -85,B 0,C 180,E1 -469.057,E2 -469.057} C_VEL
LIN {X 0,Y 608.786,Z 529.61,A -85,B 0,C 180,E1 -469.493,E2 -469.493} C_VEL
LIN {X 0,Y 608.807,Z 513.43,A -85,B 0,C 180,E1 -469.778,E2 -469.778} C_VEL
LIN {X 0,Y 608.917,Z 313.623,A -85,B 0,C 180,E1 -472.254,E2 -472.254} C_VEL
LIN {X 0,Y 608.726,Z 311.738,A -85,B 0,C 180,E1 -472.306,E2 -472.306} C_VEL
LIN {X 0,Y 608.774,Z 278.613,A -85,B 0,C 180,E1 -475.012,E2 -475.012} C_VEL
LIN {X 0,Y 608.827,Z 260.947,A -85,B 0,C 180,E1 -476.479,E2 -476.479} C_VEL
LIN {X 0,Y 608.431,Z 259.006,A -85,B 0,C 180,E1 -476.682,E2 -476.682} C_VEL
LIN {X 0,Y 608.432,Z 259.008,A -85,B 0,C 180,E1 -479.022,E2 -479.022} C_VEL
LIN {X 0,Y 608.458,Z 259.01,A -85,B 0,C 180,E1 -481.317,E2 -481.317} C_VEL
LIN {X 0,Y 608.477,Z 259.001,A -85,B 0,C 180,E1 -483.736,E2 -483.736} C_VEL
LIN {X 0,Y 608.457,Z 259,A -85,B 0,C 180,E1 -486.091,E2 -486.091} C_VEL
LIN {X 0,Y 608.458,Z 259,A -85,B 0,C 180,E1 -488.588,E2 -488.588} C_VEL
LIN {X 0,Y 608.46,Z 259.009,A -85,B 0,C 180,E1 -491.342,E2 -491.342} C_VEL
LIN {X 0,Y 608.471,Z 258.999,A -85,B 0,C 180,E1 -493.869,E2 -493.869} C_VEL
LIN {X 0,Y 608.456,Z 259.001,A -85,B 0,C 180,E1 -496.692,E2 -496.692} C_VEL
LIN {X 0,Y 608.439,Z 259.005,A -85,B 0,C 180,E1 -498.822,E2 -498.822} C_VEL
LIN {X 0,Y 608.466,Z 259,A -85,B 0,C 180,E1 -501.759,E2 -501.759} C_VEL
LIN {X 0,Y 608.439,Z 259.004,A -85,B 0,C 180,E1 -504.722,E2 -504.722} C_VEL
LIN {X 0,Y 608.46,Z 259.005,A -85,B 0,C 180,E1 -507.477,E2 -507.477} C_VEL
LIN {X 0,Y 608.466,Z 258.998,A -85,B 0,C 180,E1 -510.221,E2 -510.221} C_VEL
LIN {X 0,Y 608.47,Z 259.002,A -85,B 0,C 180,E1 -512.794,E2 -512.794} C_VEL
LIN {X 0,Y 608.452,Z 259.006,A -85,B 0,C 180,E1 -515.429,E2 -515.429} C_VEL
LIN {X 0,Y 608.461,Z 258.999,A -85,B 0,C 180,E1 -518.308,E2 -518.308} C_VEL
LIN {X 0,Y 608.451,Z 259.011,A -85,B 0,C 180,E1 -521.13,E2 -521.13} C_VEL
LIN {X 0,Y 608.459,Z 258.999,A -85,B 0,C 180,E1 -523.906,E2 -523.906} C_VEL
LIN {X 0,Y 608.458,Z 259.002,A -85,B 0,C 180,E1 -526.644,E2 -526.644} C_VEL
LIN {X 0,Y 608.462,Z 259.005,A -85,B 0,C 180,E1 -529.35,E2 -529.35} C_VEL
LIN {X 0,Y 608.477,Z 258.996,A -85,B 0,C 180,E1 -532.033,E2 -532.033} C_VEL
LIN {X 0,Y 608.459,Z 259.003,A -85,B 0,C 180,E1 -534.698,E2 -534.698} C_VEL
LIN {X 0,Y 608.473,Z 259.003,A -85,B 0,C 180,E1 -537.352,E2 -537.352} C_VEL
LIN {X 0,Y 608.477,Z 258.996,A -85,B 0,C 180,E1 -540,E2 -540} C_VEL
LIN {X 0,Y 608.468,Z 259.002,A -85,B 0,C 180,E1 -542.648,E2 -542.648} C_VEL
LIN {X 0,Y 608.464,Z 259.004,A -85,B 0,C 180,E1 -545.302,E2 -545.302} C_VEL
LIN {X 0,Y 608.478,Z 258.996,A -85,B 0,C 180,E1 -547.967,E2 -547.967} C_VEL
LIN {X 0,Y 608.458,Z 259.002,A -85,B 0,C 180,E1 -549.454,E2 -549.454} C_VEL
LIN {X 0,Y 607.779,Z 259.086,A -85,B 0,C 180,E1 -550.006,E2 -550.006} C_VEL
LIN {X 0,Y 604.926,Z 259.448,A -85,B 0,C 180,E1 -550.903,E2 -550.903} C_VEL
LIN {X 0,Y 602.524,Z 259.742,A -85,B 0,C 180,E1 -551.625,E2 -551.625} C_VEL
LIN {X 0,Y 601.491,Z 259.868,A -85,B 0,C 180,E1 -552.181,E2 -552.181} C_VEL
LIN {X 0,Y 601.407,Z 259.879,A -85,B 0,C 180,E1 -552.37,E2 -552.37} C_VEL
LIN {X 0,Y 601.425,Z 259.884,A -85,B 0,C 180,E1 -554.897,E2 -554.897} C_VEL
LIN {X 0,Y 601.428,Z 259.885,A -85,B 0,C 180,E1 -556.986,E2 -556.986} C_VEL
LIN {X 0,Y 601.403,Z 259.878,A -85,B 0,C 180,E1 -559.81,E2 -559.81} C_VEL
LIN {X 0,Y 601.41,Z 259.882,A -85,B 0,C 180,E1 -562.683,E2 -562.683} C_VEL
LIN {X 0,Y 601.4,Z 259.888,A -85,B 0,C 180,E1 -564.879,E2 -564.879} C_VEL
LIN {X 0,Y 601.414,Z 259.879,A -85,B 0,C 180,E1 -567.363,E2 -567.363} C_VEL
LIN {X 0,Y 601.427,Z 259.876,A -85,B 0,C 180,E1 -570.164,E2 -570.164} C_VEL
LIN {X 0,Y 601.417,Z 259.884,A -85,B 0,C 180,E1 -572.715,E2 -572.715} C_VEL
LIN {X 0,Y 601.411,Z 259.883,A -85,B 0,C 180,E1 -575.115,E2 -575.115} C_VEL
LIN {X 0,Y 601.432,Z 259.876,A -85,B 0,C 180,E1 -577.419,E2 -577.419} C_VEL
LIN {X 0,Y 601.402,Z 259.878,A -85,B 0,C 180,E1 -579.996,E2 -579.996} C_VEL
LIN {X 0,Y 601.41,Z 259.884,A -85,B 0,C 180,E1 -582.67,E2 -582.67} C_VEL
LIN {X 0,Y 601.425,Z 259.876,A -85,B 0,C 180,E1 -585.482,E2 -585.482} C_VEL
LIN {X 0,Y 601.424,Z 259.879,A -85,B 0,C 180,E1 -588.407,E2 -588.407} C_VEL
LIN {X 0,Y 601.434,Z 259.883,A -85,B 0,C 180,E1 -590.876,E2 -590.876} C_VEL
LIN {X 0,Y 601.397,Z 259.88,A -85,B 0,C 180,E1 -593.417,E2 -593.417} C_VEL
LIN {X 0,Y 601.432,Z 259.875,A -85,B 0,C 180,E1 -596.065,E2 -596.065} C_VEL
LIN {X 0,Y 601.418,Z 259.882,A -85,B 0,C 180,E1 -599.058,E2 -599.058} C_VEL
LIN {X 0,Y 601.415,Z 259.879,A -85,B 0,C 180,E1 -601.372,E2 -601.372} C_VEL
LIN {X 0,Y 601.395,Z 259.88,A -85,B 0,C 180,E1 -603.636,E2 -603.636} C_VEL
LIN {X 0,Y 601.399,Z 259.925,A -85,B 0,C 180,E1 -605.33,E2 -605.33} C_VEL
LIN {X 0,Y 601.991,Z 262.406,A -85,B 0,C 180,E1 -605.591,E2 -605.591} C_VEL
LIN {X 0,Y 601.882,Z 282.854,A -85,B 0,C 180,E1 -607.504,E2 -607.504} C_VEL
LIN {X 0,Y 602.346,Z 286.243,A -85,B 0,C 180,E1 -607.568,E2 -607.568} C_VEL
LIN {X 0,Y 602.134,Z 489.404,A -85,B 0,C 180,E1 -610.127,E2 -610.127} C_VEL
LIN {X 0,Y 602.081,Z 505.067,A -85,B 0,C 180,E1 -610.458,E2 -610.458} C_VEL
LIN {X 0,Y 602.012,Z 520.92,A -85,B 0,C 180,E1 -610.921,E2 -610.921} C_VEL
LIN {X 0,Y 601.905,Z 536.518,A -85,B 0,C 180,E1 -611.51,E2 -611.51} C_VEL
LIN {X 0,Y 601.85,Z 551.865,A -85,B 0,C 180,E1 -612.238,E2 -612.238} C_VEL
LIN {X 0,Y 601.767,Z 566.544,A -85,B 0,C 180,E1 -613.087,E2 -613.087} C_VEL
LIN {X 0,Y 601.67,Z 580.772,A -85,B 0,C 180,E1 -614.068,E2 -614.068} C_VEL
LIN {X 0,Y 601.601,Z 593.565,A -85,B 0,C 180,E1 -615.108,E2 -615.108} C_VEL
LIN {X 0,Y 601.526,Z 605.251,A -85,B 0,C 180,E1 -616.213,E2 -616.213} C_VEL
LIN {X 0,Y 601.463,Z 616.974,A -85,B 0,C 180,E1 -617.516,E2 -617.516} C_VEL
LIN {X 0,Y 601.41,Z 627.252,A -85,B 0,C 180,E1 -618.869,E2 -618.869} C_VEL
LIN {X 0,Y 601.393,Z 636.016,A -85,B 0,C 180,E1 -620.244,E2 -620.244} C_VEL
LIN {X 0,Y 601.364,Z 643.271,A -85,B 0,C 180,E1 -621.6,E2 -621.6} C_VEL
LIN {X 0,Y 601.364,Z 649.284,A -85,B 0,C 180,E1 -622.951,E2 -622.951} C_VEL
LIN {X 0,Y 601.349,Z 654.043,A -85,B 0,C 180,E1 -624.299,E2 -624.299} C_VEL
LIN {X 0,Y 601.342,Z 658.537,A -85,B 0,C 180,E1 -625.979,E2 -625.979} C_VEL
LIN {X 0,Y 601.312,Z 661.013,A -85,B 0,C 180,E1 -627.32,E2 -627.32} C_VEL
LIN {X 0,Y 601.342,Z 662.446,A -85,B 0,C 180,E1 -628.661,E2 -628.661} C_VEL
LIN {X 0,Y 601.332,Z 662.996,A -85,B 0,C 180,E1 -630,E2 -630} C_VEL
LIN {X 0,Y 601.339,Z 662.509,A -85,B 0,C 180,E1 -631.339,E2 -631.339} C_VEL
LIN {X 0,Y 601.312,Z 661.153,A -85,B 0,C 180,E1 -632.68,E2 -632.68} C_VEL
LIN {X 0,Y 601.339,Z 658.73,A -85,B 0,C 180,E1 -634.021,E2 -634.021} C_VEL
LIN {X 0,Y 601.346,Z 655.385,A -85,B 0,C 180,E1 -635.365,E2 -635.365} C_VEL
LIN {X 0,Y 601.364,Z 649.643,A -85,B 0,C 180,E1 -637.049,E2 -637.049} C_VEL
LIN {X 0,Y 601.366,Z 643.702,A -85,B 0,C 180,E1 -638.4,E2 -638.4} C_VEL
LIN {X 0,Y 601.387,Z 635.54,A -85,B 0,C 180,E1 -639.926,E2 -639.926} C_VEL
LIN {X 0,Y 601.428,Z 626.616,A -85,B 0,C 180,E1 -641.309,E2 -641.309} C_VEL
LIN {X 0,Y 601.472,Z 616.301,A -85,B 0,C 180,E1 -642.655,E2 -642.655} C_VEL
LIN {X 0,Y 601.533,Z 605.109,A -85,B 0,C 180,E1 -643.892,E2 -643.892} C_VEL
LIN {X 0,Y 601.594,Z 592.634,A -85,B 0,C 180,E1 -645.066,E2 -645.066} C_VEL
LIN {X 0,Y 601.655,Z 579.651,A -85,B 0,C 180,E1 -646.106,E2 -646.106} C_VEL
LIN {X 0,Y 601.755,Z 565.571,A -85,B 0,C 180,E1 -647.064,E2 -647.064} C_VEL
LIN {X 0,Y 601.866,Z 551.911,A -85,B 0,C 180,E1 -647.85,E2 -647.85} C_VEL
LIN {X 0,Y 601.94,Z 535.981,A -85,B 0,C 180,E1 -648.603,E2 -648.603} C_VEL
LIN {X 0,Y 602,Z 520.966,A -85,B 0,C 180,E1 -649.168,E2 -649.168} C_VEL
LIN {X 0,Y 602.09,Z 504.207,A -85,B 0,C 180,E1 -649.653,E2 -649.653} C_VEL
LIN {X 0,Y 602.108,Z 487.988,A -85,B 0,C 180,E1 -649.985,E2 -649.985} C_VEL
LIN {X 0,Y 602.28,Z 284.848,A -85,B 0,C 180,E1 -652.542,E2 -652.542} C_VEL
LIN {X 0,Y 601.876,Z 282.541,A -85,B 0,C 180,E1 -652.616,E2 -652.616} C_VEL
LIN {X 0,Y 601.881,Z 261.798,A -85,B 0,C 180,E1 -654.561,E2 -654.561} C_VEL
LIN {X 0,Y 601.38,Z 259.887,A -85,B 0,C 180,E1 -654.768,E2 -654.768} C_VEL
LIN {X 0,Y 601.411,Z 259.888,A -85,B 0,C 180,E1 -657.362,E2 -657.362} C_VEL
LIN {X 0,Y 601.428,Z 259.876,A -85,B 0,C 180,E1 -660.164,E2 -660.164} C_VEL
LIN {X 0,Y 601.409,Z 259.879,A -85,B 0,C 180,E1 -662.713,E2 -662.713} C_VEL
LIN {X 0,Y 601.386,Z 259.888,A -85,B 0,C 180,E1 -665.111,E2 -665.111} C_VEL
LIN {X 0,Y 601.434,Z 259.883,A -85,B 0,C 180,E1 -667.419,E2 -667.419} C_VEL
LIN {X 0,Y 601.4,Z 259.879,A -85,B 0,C 180,E1 -669.995,E2 -669.995} C_VEL
LIN {X 0,Y 601.405,Z 259.879,A -85,B 0,C 180,E1 -672.67,E2 -672.67} C_VEL
LIN {X 0,Y 601.424,Z 259.882,A -85,B 0,C 180,E1 -675.482,E2 -675.482} C_VEL
LIN {X 0,Y 601.417,Z 259.876,A -85,B 0,C 180,E1 -678.407,E2 -678.407} C_VEL
LIN {X 0,Y 601.408,Z 259.882,A -85,B 0,C 180,E1 -680.873,E2 -680.873} C_VEL
LIN {X 0,Y 601.441,Z 259.876,A -85,B 0,C 180,E1 -683.734,E2 -683.734} C_VEL
LIN {X 0,Y 601.412,Z 259.879,A -85,B 0,C 180,E1 -686.686,E2 -686.686} C_VEL
LIN {X 0,Y 601.414,Z 259.885,A -85,B 0,C 180,E1 -689.058,E2 -689.058} C_VEL
LIN {X 0,Y 601.431,Z 259.881,A -85,B 0,C 180,E1 -691.373,E2 -691.373} C_VEL
LIN {X 0,Y 601.399,Z 259.881,A -85,B 0,C 180,E1 -693.636,E2 -693.636} C_VEL
LIN {X 0,Y 601.417,Z 259.878,A -85,B 0,C 180,E1 -696.59,E2 -696.59} C_VEL
LIN {X 0,Y 601.429,Z 259.879,A -85,B 0,C 180,E1 -699.478,E2 -699.478} C_VEL
LIN {X 0,Y 601.394,Z 259.879,A -85,B 0,C 180,E1 -702.312,E2 -702.312} C_VEL
LIN {X 0,Y 601.41,Z 259.877,A -85,B 0,C 180,E1 -704.409,E2 -704.409} C_VEL
LIN {X 0,Y 601.415,Z 259.885,A -85,B 0,C 180,E1 -707.172,E2 -707.172} C_VEL
LIN {X 0,Y 601.432,Z 259.874,A -85,B 0,C 180,E1 -709.905,E2 -709.905} C_VEL
LIN {X 0,Y 601.438,Z 259.877,A -85,B 0,C 180,E1 -712.615,E2 -712.615} C_VEL
LIN {X 0,Y 601.416,Z 259.882,A -85,B 0,C 180,E1 -715.308,E2 -715.308} C_VEL
LIN {X 0,Y 601.435,Z 259.873,A -85,B 0,C 180,E1 -717.991,E2 -717.991} C_VEL
LIN {X 0,Y 601.445,Z 259.878,A -85,B 0,C 180,E1 -720.669,E2 -720.669} C_VEL
LIN {X 0,Y 601.426,Z 259.878,A -85,B 0,C 180,E1 -723.349,E2 -723.349} C_VEL
LIN {X 0,Y 601.435,Z 259.874,A -85,B 0,C 180,E1 -726.037,E2 -726.037} C_VEL
LIN {X 0,Y 601.41,Z 259.884,A -85,B 0,C 180,E1 -728.738,E2 -728.738} C_VEL
LIN {X 0,Y 601.432,Z 259.876,A -85,B 0,C 180,E1 -731.458,E2 -731.458} C_VEL
LIN {X 0,Y 601.416,Z 259.877,A -85,B 0,C 180,E1 -734.205,E2 -734.205} C_VEL
LIN {X 0,Y 601.427,Z 259.884,A -85,B 0,C 180,E1 -736.986,E2 -736.986} C_VEL
LIN {X 0,Y 601.401,Z 259.878,A -85,B 0,C 180,E1 -739.809,E2 -739.809} C_VEL
LIN {X 0,Y 601.412,Z 259.883,A -85,B 0,C 180,E1 -742.606,E2 -742.606} C_VEL
LIN {X 0,Y 601.399,Z 259.89,A -85,B 0,C 180,E1 -744.879,E2 -744.879} C_VEL
LIN {X 0,Y 601.41,Z 259.88,A -85,B 0,C 180,E1 -747.362,E2 -747.362} C_VEL
LIN {X 0,Y 601.425,Z 259.876,A -85,B 0,C 180,E1 -750.164,E2 -750.164} C_VEL
LIN {X 0,Y 601.418,Z 259.885,A -85,B 0,C 180,E1 -752.716,E2 -752.716} C_VEL
LIN {X 0,Y 601.413,Z 259.882,A -85,B 0,C 180,E1 -755.115,E2 -755.115} C_VEL
LIN {X 0,Y 601.43,Z 259.876,A -85,B 0,C 180,E1 -757.419,E2 -757.419} C_VEL
LIN {X 0,Y 601.401,Z 259.879,A -85,B 0,C 180,E1 -759.996,E2 -759.996} C_VEL
LIN {X 0,Y 601.407,Z 259.887,A -85,B 0,C 180,E1 -762.67,E2 -762.67} C_VEL
LIN {X 0,Y 601.423,Z 259.876,A -85,B 0,C 180,E1 -765.482,E2 -765.482} C_VEL
LIN {X 0,Y 601.424,Z 259.881,A -85,B 0,C 180,E1 -768.407,E2 -768.407} C_VEL
LIN {X 0,Y 601.424,Z 259.883,A -85,B 0,C 180,E1 -770.875,E2 -770.875} C_VEL
LIN {X 0,Y 601.397,Z 259.88,A -85,B 0,C 180,E1 -773.417,E2 -773.417} C_VEL
LIN {X 0,Y 601.432,Z 259.875,A -85,B 0,C 180,E1 -776.064,E2 -776.064} C_VEL
LIN {X 0,Y 601.415,Z 259.881,A -85,B 0,C 180,E1 -779.058,E2 -779.058} C_VEL
LIN {X 0,Y 601.411,Z 259.879,A -85,B 0,C 180,E1 -781.372,E2 -781.372} C_VEL
LIN {X 0,Y 601.432,Z 259.981,A -85,B 0,C 180,E1 -783.088,E2 -783.088} C_VEL
LIN {X 0,Y 602.18,Z 263.156,A -85,B 0,C 180,E1 -783.393,E2 -783.393} C_VEL
LIN {X 0,Y 602.029,Z 295.176,A -85,B 0,C 180,E1 -786.067,E2 -786.067} C_VEL
LIN {X 0,Y 601.96,Z 312.019,A -85,B 0,C 180,E1 -787.453,E2 -787.453} C_VEL
LIN {X 0,Y 602.355,Z 315.853,A -85,B 0,C 180,E1 -787.519,E2 -787.519} C_VEL
LIN {X 0,Y 602.124,Z 517.951,A -85,B 0,C 180,E1 -790.06,E2 -790.06} C_VEL
LIN {X 0,Y 602.075,Z 534.181,A -85,B 0,C 180,E1 -790.391,E2 -790.391} C_VEL
LIN {X 0,Y 602.011,Z 550.944,A -85,B 0,C 180,E1 -790.877,E2 -790.877} C_VEL
LIN {X 0,Y 601.915,Z 566.241,A -85,B 0,C 180,E1 -791.453,E2 -791.453} C_VEL
LIN {X 0,Y 601.868,Z 581.016,A -85,B 0,C 180,E1 -792.151,E2 -792.151} C_VEL
LIN {X 0,Y 601.767,Z 594.845,A -85,B 0,C 180,E1 -792.937,E2 -792.937} C_VEL
LIN {X 0,Y 601.696,Z 609.051,A -85,B 0,C 180,E1 -793.895,E2 -793.895} C_VEL
LIN {X 0,Y 601.592,Z 622.128,A -85,B 0,C 180,E1 -794.934,E2 -794.934} C_VEL
LIN {X 0,Y 601.555,Z 634.679,A -85,B 0,C 180,E1 -796.108,E2 -796.108} C_VEL
LIN {X 0,Y 601.472,Z 645.912,A -85,B 0,C 180,E1 -797.345,E2 -797.345} C_VEL
LIN {X 0,Y 601.427,Z 656.287,A -85,B 0,C 180,E1 -798.691,E2 -798.691} C_VEL
LIN {X 0,Y 601.387,Z 665.272,A -85,B 0,C 180,E1 -800.074,E2 -800.074} C_VEL
LIN {X 0,Y 601.365,Z 673.487,A -85,B 0,C 180,E1 -801.6,E2 -801.6} C_VEL
LIN {X 0,Y 601.362,Z 679.468,A -85,B 0,C 180,E1 -802.951,E2 -802.951} C_VEL
LIN {X 0,Y 601.345,Z 685.246,A -85,B 0,C 180,E1 -804.635,E2 -804.635} C_VEL
LIN {X 0,Y 601.34,Z 688.633,A -85,B 0,C 180,E1 -805.979,E2 -805.979} C_VEL
LIN {X 0,Y 601.311,Z 691.086,A -85,B 0,C 180,E1 -807.32,E2 -807.32} C_VEL
LIN {X 0,Y 601.34,Z 692.477,A -85,B 0,C 180,E1 -808.661,E2 -808.661} C_VEL
LIN {X 0,Y 601.33,Z 693,A -85,B 0,C 180,E1 -810,E2 -810} C_VEL
LIN {X 0,Y 601.34,Z 692.477,A -85,B 0,C 180,E1 -811.339,E2 -811.339} C_VEL
LIN {X 0,Y 601.311,Z 691.086,A -85,B 0,C 180,E1 -812.68,E2 -812.68} C_VEL
LIN {X 0,Y 601.34,Z 688.633,A -85,B 0,C 180,E1 -814.021,E2 -814.021} C_VEL
LIN {X 0,Y 601.345,Z 685.246,A -85,B 0,C 180,E1 -815.365,E2 -815.365} C_VEL
LIN {X 0,Y 601.362,Z 679.469,A -85,B 0,C 180,E1 -817.049,E2 -817.049} C_VEL
LIN {X 0,Y 601.376,Z 671.858,A -85,B 0,C 180,E1 -818.738,E2 -818.738} C_VEL
LIN {X 0,Y 601.411,Z 663.246,A -85,B 0,C 180,E1 -820.265,E2 -820.265} C_VEL
LIN {X 0,Y 601.429,Z 653.969,A -85,B 0,C 180,E1 -821.629,E2 -821.629} C_VEL
LIN {X 0,Y 601.479,Z 644.423,A -85,B 0,C 180,E1 -822.827,E2 -822.827} C_VEL
LIN {X 0,Y 601.544,Z 633.62,A -85,B 0,C 180,E1 -823.997,E2 -823.997} C_VEL
LIN {X 0,Y 601.606,Z 621.144,A -85,B 0,C 180,E1 -825.152,E2 -825.152} C_VEL
LIN {X 0,Y 601.707,Z 607.886,A -85,B 0,C 180,E1 -826.192,E2 -826.192} C_VEL
LIN {X 0,Y 601.787,Z 593.433,A -85,B 0,C 180,E1 -827.15,E2 -827.15} C_VEL
LIN {X 0,Y 601.863,Z 579.266,A -85,B 0,C 180,E1 -827.938,E2 -827.938} C_VEL
LIN {X 0,Y 601.942,Z 564.913,A -85,B 0,C 180,E1 -828.604,E2 -828.604} C_VEL
LIN {X 0,Y 602.011,Z 548.35,A -85,B 0,C 180,E1 -829.212,E2 -829.212} C_VEL
LIN {X 0,Y 602.09,Z 532.354,A -85,B 0,C 180,E1 -829.653,E2 -829.653} C_VEL
LIN {X 0,Y 602.142,Z 516.443,A -85,B 0,C 180,E1 -829.962,E2 -829.962} C_VEL
LIN {X 0,Y 602.32,Z 314.081,A -85,B 0,C 180,E1 -832.505,E2 -832.505} C_VEL
LIN {X 0,Y 601.968,Z 311.814,A -85,B 0,C 180,E1 -832.564,E2 -832.564} C_VEL
LIN {X 0,Y 602.109,Z 277.509,A -85,B 0,C 180,E1 -835.401,E2 -835.401} C_VEL
LIN {X 0,Y 602.179,Z 263.155,A -85,B 0,C 180,E1 -836.607,E2 -836.607} C_VEL
LIN {X 0,Y 601.407,Z 259.886,A -85,B 0,C 180,E1 -836.925,E2 -836.925} C_VEL
LIN {X 0,Y 601.406,Z 259.888,A -85,B 0,C 180,E1 -839.394,E2 -839.394} C_VEL
LIN {X 0,Y 601.402,Z 259.883,A -85,B 0,C 180,E1 -841.727,E2 -841.727} C_VEL
LIN {X 0,Y 601.424,Z 259.876,A -85,B 0,C 180,E1 -844.118,E2 -844.118} C_VEL
LIN {X 0,Y 601.397,Z 259.88,A -85,B 0,C 180,E1 -846.583,E2 -846.583} C_VEL
LIN {X 0,Y 601.436,Z 259.88,A -85,B 0,C 180,E1 -849.535,E2 -849.535} C_VEL
LIN {X 0,Y 601.404,Z 259.879,A -85,B 0,C 180,E1 -852.59,E2 -852.59} C_VEL
LIN {X 0,Y 601.422,Z 259.876,A -85,B 0,C 180,E1 -854.535,E2 -854.535} C_VEL
LIN {X 0,Y 601.409,Z 259.885,A -85,B 0,C 180,E1 -857.409,E2 -857.409} C_VEL
LIN {X 0,Y 601.402,Z 259.878,A -85,B 0,C 180,E1 -860.004,E2 -860.004} C_VEL
LIN {X 0,Y 601.43,Z 259.876,A -85,B 0,C 180,E1 -862.618,E2 -862.618} C_VEL
LIN {X 0,Y 601.418,Z 259.884,A -85,B 0,C 180,E1 -865.068,E2 -865.068} C_VEL
LIN {X 0,Y 601.429,Z 259.88,A -85,B 0,C 180,E1 -867.484,E2 -867.484} C_VEL
LIN {X 0,Y 601.426,Z 259.876,A -85,B 0,C 180,E1 -869.851,E2 -869.851} C_VEL
LIN {X 0,Y 601.409,Z 259.879,A -85,B 0,C 180,E1 -872.638,E2 -872.638} C_VEL
LIN {X 0,Y 601.398,Z 259.889,A -85,B 0,C 180,E1 -875.121,E2 -875.121} C_VEL
LIN {X 0,Y 601.412,Z 259.883,A -85,B 0,C 180,E1 -877.394,E2 -877.394} C_VEL
LIN {X 0,Y 601.401,Z 259.877,A -85,B 0,C 180,E1 -880.191,E2 -880.191} C_VEL
LIN {X 0,Y 601.428,Z 259.884,A -85,B 0,C 180,E1 -883.014,E2 -883.014} C_VEL
LIN {X 0,Y 601.419,Z 259.875,A -85,B 0,C 180,E1 -885.908,E2 -885.908} C_VEL
LIN {X 0,Y 601.431,Z 259.876,A -85,B 0,C 180,E1 -888.542,E2 -888.542} C_VEL
LIN {X 0,Y 601.411,Z 259.884,A -85,B 0,C 180,E1 -891.262,E2 -891.262} C_VEL
LIN {X 0,Y 601.435,Z 259.873,A -85,B 0,C 180,E1 -893.963,E2 -893.963} C_VEL
LIN {X 0,Y 601.424,Z 259.879,A -85,B 0,C 180,E1 -896.651,E2 -896.651} C_VEL
LIN {X 0,Y 601.448,Z 259.877,A -85,B 0,C 180,E1 -899.331,E2 -899.331} C_VEL
LIN {X 0,Y 601.435,Z 259.873,A -85,B 0,C 180,E1 -902.009,E2 -902.009} C_VEL
LIN {X 0,Y 601.415,Z 259.881,A -85,B 0,C 180,E1 -904.692,E2 -904.692} C_VEL
LIN {X 0,Y 601.44,Z 259.876,A -85,B 0,C 180,E1 -907.385,E2 -907.385} C_VEL
LIN {X 0,Y 601.432,Z 259.874,A -85,B 0,C 180,E1 -910.095,E2 -910.095} C_VEL
LIN {X 0,Y 601.407,Z 259.879,A -85,B 0,C 180,E1 -912.37,E2 -912.37} C_VEL
LIN {X 0,Y 600.739,Z 259.971,A -85,B 0,C 180,E1 -912.929,E2 -912.929} C_VEL
LIN {X 0,Y 597.889,Z 260.328,A -85,B 0,C 180,E1 -913.837,E2 -913.837} C_VEL
LIN {X 0,Y 595.48,Z 260.627,A -85,B 0,C 180,E1 -914.567,E2 -914.567} C_VEL
LIN {X 0,Y 594.443,Z 260.751,A -85,B 0,C 180,E1 -915.131,E2 -915.131} C_VEL
LIN {X 0,Y 594.358,Z 260.759,A -85,B 0,C 180,E1 -915.321,E2 -915.321} C_VEL
LIN {X 0,Y 594.353,Z 260.756,A -85,B 0,C 180,E1 -917.905,E2 -917.905} C_VEL
LIN {X 0,Y 594.4,Z 260.758,A -85,B 0,C 180,E1 -920.776,E2 -920.776} C_VEL
LIN {X 0,Y 594.39,Z 260.752,A -85,B 0,C 180,E1 -923.704,E2 -923.704} C_VEL
LIN {X 0,Y 594.382,Z 260.759,A -85,B 0,C 180,E1 -926.7,E2 -926.7} C_VEL
LIN {X 0,Y 594.379,Z 260.762,A -85,B 0,C 180,E1 -928.999,E2 -928.999} C_VEL
LIN {X 0,Y 594.374,Z 260.754,A -85,B 0,C 180,E1 -931.643,E2 -931.643} C_VEL
LIN {X 0,Y 594.395,Z 260.756,A -85,B 0,C 180,E1 -934.579,E2 -934.579} C_VEL
LIN {X 0,Y 594.383,Z 260.758,A -85,B 0,C 180,E1 -937.087,E2 -937.087} C_VEL
LIN {X 0,Y 594.357,Z 260.756,A -85,B 0,C 180,E1 -939.773,E2 -939.773} C_VEL
LIN {X 0,Y 594.368,Z 260.757,A -85,B 0,C 180,E1 -942.376,E2 -942.376} C_VEL
LIN {X 0,Y 594.363,Z 260.759,A -85,B 0,C 180,E1 -945.191,E2 -945.191} C_VEL
LIN {X 0,Y 594.365,Z 260.755,A -85,B 0,C 180,E1 -947.625,E2 -947.625} C_VEL
LIN {X 0,Y 594.391,Z 260.755,A -85,B 0,C 180,E1 -950.321,E2 -950.321} C_VEL
LIN {X 0,Y 594.381,Z 260.761,A -85,B 0,C 180,E1 -952.913,E2 -952.913} C_VEL
LIN {X 0,Y 594.378,Z 260.753,A -85,B 0,C 180,E1 -955.862,E2 -955.862} C_VEL
LIN {X 0,Y 594.378,Z 260.762,A -85,B 0,C 180,E1 -958.65,E2 -958.65} C_VEL
LIN {X 0,Y 594.376,Z 260.76,A -85,B 0,C 180,E1 -961.043,E2 -961.043} C_VEL
LIN {X 0,Y 594.379,Z 260.757,A -85,B 0,C 180,E1 -963.3,E2 -963.3} C_VEL
LIN {X 0,Y 594.392,Z 260.892,A -85,B 0,C 180,E1 -965.112,E2 -965.112} C_VEL
LIN {X 0,Y 595.232,Z 265.505,A -85,B 0,C 180,E1 -965.591,E2 -965.591} C_VEL
LIN {X 0,Y 595.086,Z 282.813,A -85,B 0,C 180,E1 -967.228,E2 -967.228} C_VEL
LIN {X 0,Y 595.758,Z 286.277,A -85,B 0,C 180,E1 -967.306,E2 -967.306} C_VEL
LIN {X 0,Y 595.453,Z 487.949,A -85,B 0,C 180,E1 -969.872,E2 -969.872} C_VEL
LIN {X 0,Y 595.388,Z 503.267,A -85,B 0,C 180,E1 -970.184,E2 -970.184} C_VEL
LIN {X 0,Y 595.272,Z 519.643,A -85,B 0,C 180,E1 -970.651,E2 -970.651} C_VEL
LIN {X 0,Y 595.173,Z 535.484,A -85,B 0,C 180,E1 -971.246,E2 -971.246} C_VEL
LIN {X 0,Y 595.042,Z 551.88,A -85,B 0,C 180,E1 -972.028,E2 -972.028} C_VEL
LIN {X 0,Y 594.898,Z 565.541,A -85,B 0,C 180,E1 -972.822,E2 -972.822} C_VEL
LIN {X 0,Y 594.795,Z 579.621,A -85,B 0,C 180,E1 -973.791,E2 -973.791} C_VEL
LIN {X 0,Y 594.648,Z 591.625,A -85,B 0,C 180,E1 -974.754,E2 -974.754} C_VEL
LIN {X 0,Y 594.579,Z 603.872,A -85,B 0,C 180,E1 -975.905,E2 -975.905} C_VEL
LIN {X 0,Y 594.449,Z 615.526,A -85,B 0,C 180,E1 -977.193,E2 -977.193} C_VEL
LIN {X 0,Y 594.408,Z 624.887,A -85,B 0,C 180,E1 -978.405,E2 -978.405} C_VEL
LIN {X 0,Y 594.369,Z 633.996,A -85,B 0,C 180,E1 -979.784,E2 -979.784} C_VEL
LIN {X 0,Y 594.319,Z 641.623,A -85,B 0,C 180,E1 -981.157,E2 -981.157} C_VEL
LIN {X 0,Y 594.276,Z 647.862,A -85,B 0,C 180,E1 -982.525,E2 -982.525} C_VEL
LIN {X 0,Y 594.254,Z 652.983,A -85,B 0,C 180,E1 -983.89,E2 -983.89} C_VEL
LIN {X 0,Y 594.23,Z 656.939,A -85,B 0,C 180,E1 -985.251,E2 -985.251} C_VEL
LIN {X 0,Y 594.253,Z 659.909,A -85,B 0,C 180,E1 -986.61,E2 -986.61} C_VEL
LIN {X 0,Y 594.239,Z 661.838,A -85,B 0,C 180,E1 -987.967,E2 -987.967} C_VEL
LIN {X 0,Y 594.235,Z 662.84,A -85,B 0,C 180,E1 -989.322,E2 -989.322} C_VEL
LIN {X 0,Y 594.235,Z 662.861,A -85,B 0,C 180,E1 -990.678,E2 -990.678} C_VEL
LIN {X 0,Y 594.239,Z 661.942,A -85,B 0,C 180,E1 -992.033,E2 -992.033} C_VEL
LIN {X 0,Y 594.255,Z 660.057,A -85,B 0,C 180,E1 -993.39,E2 -993.39} C_VEL
LIN {X 0,Y 594.226,Z 657.174,A -85,B 0,C 180,E1 -994.749,E2 -994.749} C_VEL
LIN {X 0,Y 594.257,Z 653.264,A -85,B 0,C 180,E1 -996.11,E2 -996.11} C_VEL
LIN {X 0,Y 594.276,Z 648.237,A -85,B 0,C 180,E1 -997.475,E2 -997.475} C_VEL
LIN {X 0,Y 594.317,Z 642.081,A -85,B 0,C 180,E1 -998.843,E2 -998.843} C_VEL
LIN {X 0,Y 594.36,Z 633.513,A -85,B 0,C 180,E1 -1000.388,E2 -1000.388} C_VEL
LIN {X 0,Y 594.407,Z 624.293,A -85,B 0,C 180,E1 -1001.768,E2 -1001.768} C_VEL
LIN {X 0,Y 594.467,Z 614.81,A -85,B 0,C 180,E1 -1002.981,E2 -1002.981} C_VEL
LIN {X 0,Y 594.559,Z 603.333,A -85,B 0,C 180,E1 -1004.238,E2 -1004.238} C_VEL
LIN {X 0,Y 594.665,Z 590.639,A -85,B 0,C 180,E1 -1005.421,E2 -1005.421} C_VEL
LIN {X 0,Y 594.783,Z 577.31,A -85,B 0,C 180,E1 -1006.474,E2 -1006.474} C_VEL
LIN {X 0,Y 594.924,Z 564.154,A -85,B 0,C 180,E1 -1007.354,E2 -1007.354} C_VEL
LIN {X 0,Y 595.04,Z 550.156,A -85,B 0,C 180,E1 -1008.15,E2 -1008.15} C_VEL
LIN {X 0,Y 595.19,Z 535.233,A -85,B 0,C 180,E1 -1008.854,E2 -1008.854} C_VEL
LIN {X 0,Y 595.299,Z 518.355,A -85,B 0,C 180,E1 -1009.482,E2 -1009.482} C_VEL
LIN {X 0,Y 595.385,Z 502.358,A -85,B 0,C 180,E1 -1009.928,E2 -1009.928} C_VEL
LIN {X 0,Y 595.449,Z 484.937,A -85,B 0,C 180,E1 -1010.263,E2 -1010.263} C_VEL
LIN {X 0,Y 595.75,Z 286.177,A -85,B 0,C 180,E1 -1012.785,E2 -1012.785} C_VEL
LIN {X 0,Y 595.106,Z 282.729,A -85,B 0,C 180,E1 -1012.869,E2 -1012.869} C_VEL
LIN {X 0,Y 595.195,Z 264.424,A -85,B 0,C 180,E1 -1014.604,E2 -1014.604} C_VEL
LIN {X 0,Y 594.348,Z 260.766,A -85,B 0,C 180,E1 -1015.015,E2 -1015.015} C_VEL
LIN {X 0,Y 594.367,Z 260.763,A -85,B 0,C 180,E1 -1017.523,E2 -1017.523} C_VEL
LIN {X 0,Y 594.385,Z 260.753,A -85,B 0,C 180,E1 -1020.328,E2 -1020.328} C_VEL
LIN {X 0,Y 594.375,Z 260.758,A -85,B 0,C 180,E1 -1022.95,E2 -1022.95} C_VEL
LIN {X 0,Y 594.347,Z 260.765,A -85,B 0,C 180,E1 -1025.409,E2 -1025.409} C_VEL
LIN {X 0,Y 594.382,Z 260.754,A -85,B 0,C 180,E1 -1027.941,E2 -1027.941} C_VEL
LIN {X 0,Y 594.373,Z 260.757,A -85,B 0,C 180,E1 -1030.821,E2 -1030.821} C_VEL
LIN {X 0,Y 594.381,Z 260.755,A -85,B 0,C 180,E1 -1033.841,E2 -1033.841} C_VEL
LIN {X 0,Y 594.364,Z 260.757,A -85,B 0,C 180,E1 -1036.7,E2 -1036.7} C_VEL
LIN {X 0,Y 594.37,Z 260.761,A -85,B 0,C 180,E1 -1039.433,E2 -1039.433} C_VEL
LIN {X 0,Y 594.386,Z 260.752,A -85,B 0,C 180,E1 -1042.391,E2 -1042.391} C_VEL
LIN {X 0,Y 594.356,Z 260.758,A -85,B 0,C 180,E1 -1044.675,E2 -1044.675} C_VEL
LIN {X 0,Y 594.375,Z 260.762,A -85,B 0,C 180,E1 -1047.088,E2 -1047.088} C_VEL
LIN {X 0,Y 594.384,Z 260.755,A -85,B 0,C 180,E1 -1049.671,E2 -1049.671} C_VEL
LIN {X 0,Y 594.372,Z 260.754,A -85,B 0,C 180,E1 -1052.539,E2 -1052.539} C_VEL
LIN {X 0,Y 594.37,Z 260.759,A -85,B 0,C 180,E1 -1054.807,E2 -1054.807} C_VEL
LIN {X 0,Y 594.362,Z 260.762,A -85,B 0,C 180,E1 -1057.264,E2 -1057.264} C_VEL
LIN {X 0,Y 594.371,Z 260.754,A -85,B 0,C 180,E1 -1059.946,E2 -1059.946} C_VEL
LIN {X 0,Y 594.386,Z 260.757,A -85,B 0,C 180,E1 -1062.806,E2 -1062.806} C_VEL
LIN {X 0,Y 594.387,Z 260.753,A -85,B 0,C 180,E1 -1065.826,E2 -1065.826} C_VEL
LIN {X 0,Y 594.392,Z 260.753,A -85,B 0,C 180,E1 -1068.404,E2 -1068.404} C_VEL
LIN {X 0,Y 594.377,Z 260.761,A -85,B 0,C 180,E1 -1071.158,E2 -1071.158} C_VEL
LIN {X 0,Y 594.389,Z 260.752,A -85,B 0,C 180,E1 -1073.891,E2 -1073.891} C_VEL
LIN {X 0,Y 594.378,Z 260.756,A -85,B 0,C 180,E1 -1076.611,E2 -1076.611} C_VEL
LIN {X 0,Y 594.417,Z 260.753,A -85,B 0,C 180,E1 -1079.322,E2 -1079.322} C_VEL
LIN {X 0,Y 594.403,Z 260.75,A -85,B 0,C 180,E1 -1082.033,E2 -1082.033} C_VEL
LIN {X 0,Y 594.386,Z 260.757,A -85,B 0,C 180,E1 -1084.748,E2 -1084.748} C_VEL
LIN {X 0,Y 594.391,Z 260.754,A -85,B 0,C 180,E1 -1087.473,E2 -1087.473} C_VEL
LIN {X 0,Y 594.392,Z 260.751,A -85,B 0,C 180,E1 -1090.216,E2 -1090.216} C_VEL
LIN {X 0,Y 594.363,Z 260.765,A -85,B 0,C 180,E1 -1092.983,E2 -1092.983} C_VEL
LIN {X 0,Y 594.369,Z 260.762,A -85,B 0,C 180,E1 -1095.078,E2 -1095.078} C_VEL
LIN {X 0,Y 594.386,Z 260.758,A -85,B 0,C 180,E1 -1097.193,E2 -1097.193} C_VEL
LIN {X 0,Y 594.372,Z 260.754,A -85,B 0,C 180,E1 -1100.054,E2 -1100.054} C_VEL
LIN {X 0,Y 594.361,Z 260.764,A -85,B 0,C 180,E1 -1102.967,E2 -1102.967} C_VEL
LIN {X 0,Y 594.37,Z 260.759,A -85,B 0,C 180,E1 -1105.193,E2 -1105.193} C_VEL
LIN {X 0,Y 594.382,Z 260.754,A -85,B 0,C 180,E1 -1107.527,E2 -1107.527} C_VEL
LIN {X 0,Y 594.383,Z 260.755,A -85,B 0,C 180,E1 -1110.328,E2 -1110.328} C_VEL
LIN {X 0,Y 594.373,Z 260.762,A -85,B 0,C 180,E1 -1112.95,E2 -1112.95} C_VEL
LIN {X 0,Y 594.38,Z 260.755,A -85,B 0,C 180,E1 -1115.407,E2 -1115.407} C_VEL
LIN {X 0,Y 594.385,Z 260.753,A -85,B 0,C 180,E1 -1117.941,E2 -1117.941} C_VEL
LIN {X 0,Y 594.381,Z 260.763,A -85,B 0,C 180,E1 -1120.823,E2 -1120.823} C_VEL
LIN {X 0,Y 594.364,Z 260.755,A -85,B 0,C 180,E1 -1123.84,E2 -1123.84} C_VEL
LIN {X 0,Y 594.376,Z 260.764,A -85,B 0,C 180,E1 -1126.702,E2 -1126.702} C_VEL
LIN {X 0,Y 594.365,Z 260.756,A -85,B 0,C 180,E1 -1129.433,E2 -1129.433} C_VEL
LIN {X 0,Y 594.386,Z 260.758,A -85,B 0,C 180,E1 -1132.392,E2 -1132.392} C_VEL
LIN {X 0,Y 594.371,Z 260.754,A -85,B 0,C 180,E1 -1135.42,E2 -1135.42} C_VEL
LIN {X 0,Y 594.38,Z 260.758,A -85,B 0,C 180,E1 -1138.357,E2 -1138.357} C_VEL
LIN {X 0,Y 594.374,Z 260.76,A -85,B 0,C 180,E1 -1141.043,E2 -1141.043} C_VEL
LIN {X 0,Y 594.419,Z 260.947,A -85,B 0,C 180,E1 -1142.828,E2 -1142.828} C_VEL
LIN {X 0,Y 595.551,Z 265.364,A -85,B 0,C 180,E1 -1143.263,E2 -1143.263} C_VEL
LIN {X 0,Y 595.275,Z 298.489,A -85,B 0,C 180,E1 -1146.056,E2 -1146.056} C_VEL
LIN {X 0,Y 595.274,Z 312.409,A -85,B 0,C 180,E1 -1147.192,E2 -1147.192} C_VEL
LIN {X 0,Y 595.796,Z 317.088,A -85,B 0,C 180,E1 -1147.273,E2 -1147.273} C_VEL
LIN {X 0,Y 595.471,Z 517.951,A -85,B 0,C 180,E1 -1149.827,E2 -1149.827} C_VEL
LIN {X 0,Y 595.406,Z 534.182,A -85,B 0,C 180,E1 -1150.163,E2 -1150.163} C_VEL
LIN {X 0,Y 595.27,Z 550.947,A -85,B 0,C 180,E1 -1150.651,E2 -1150.651} C_VEL
LIN {X 0,Y 595.153,Z 566.488,A -85,B 0,C 180,E1 -1151.245,E2 -1151.245} C_VEL
LIN {X 0,Y 595.055,Z 581.019,A -85,B 0,C 180,E1 -1151.939,E2 -1151.939} C_VEL
LIN {X 0,Y 594.909,Z 594.848,A -85,B 0,C 180,E1 -1152.734,E2 -1152.734} C_VEL
LIN {X 0,Y 594.812,Z 609.054,A -85,B 0,C 180,E1 -1153.703,E2 -1153.703} C_VEL
LIN {X 0,Y 594.647,Z 622.127,A -85,B 0,C 180,E1 -1154.754,E2 -1154.754} C_VEL
LIN {X 0,Y 594.558,Z 634.316,A -85,B 0,C 180,E1 -1155.904,E2 -1155.904} C_VEL
LIN {X 0,Y 594.449,Z 645.911,A -85,B 0,C 180,E1 -1157.193,E2 -1157.193} C_VEL
LIN {X 0,Y 594.381,Z 656.424,A -85,B 0,C 180,E1 -1158.574,E2 -1158.574} C_VEL
LIN {X 0,Y 594.334,Z 665.273,A -85,B 0,C 180,E1 -1159.955,E2 -1159.955} C_VEL
LIN {X 0,Y 594.295,Z 673.487,A -85,B 0,C 180,E1 -1161.499,E2 -1161.499} C_VEL
LIN {X 0,Y 594.284,Z 679.468,A -85,B 0,C 180,E1 -1162.867,E2 -1162.867} C_VEL
LIN {X 0,Y 594.263,Z 685.246,A -85,B 0,C 180,E1 -1164.571,E2 -1164.571} C_VEL
LIN {X 0,Y 594.253,Z 688.634,A -85,B 0,C 180,E1 -1165.931,E2 -1165.931} C_VEL
LIN {X 0,Y 594.213,Z 691.087,A -85,B 0,C 180,E1 -1167.288,E2 -1167.288} C_VEL
LIN {X 0,Y 594.24,Z 692.478,A -85,B 0,C 180,E1 -1168.645,E2 -1168.645} C_VEL
LIN {X 0,Y 594.231,Z 693,A -85,B 0,C 180,E1 -1170,E2 -1170} C_VEL
LIN {X 0,Y 594.24,Z 692.478,A -85,B 0,C 180,E1 -1171.355,E2 -1171.355} C_VEL
LIN {X 0,Y 594.213,Z 691.087,A -85,B 0,C 180,E1 -1172.712,E2 -1172.712} C_VEL
LIN {X 0,Y 594.253,Z 688.634,A -85,B 0,C 180,E1 -1174.069,E2 -1174.069} C_VEL
LIN {X 0,Y 594.279,Z 684.186,A -85,B 0,C 180,E1 -1175.769,E2 -1175.769} C_VEL
LIN {X 0,Y 594.284,Z 679.469,A -85,B 0,C 180,E1 -1177.133,E2 -1177.133} C_VEL
LIN {X 0,Y 594.318,Z 671.857,A -85,B 0,C 180,E1 -1178.843,E2 -1178.843} C_VEL
LIN {X 0,Y 594.354,Z 663.248,A -85,B 0,C 180,E1 -1180.389,E2 -1180.389} C_VEL
LIN {X 0,Y 594.406,Z 653.97,A -85,B 0,C 180,E1 -1181.768,E2 -1181.768} C_VEL
LIN {X 0,Y 594.469,Z 644.424,A -85,B 0,C 180,E1 -1182.981,E2 -1182.981} C_VEL
LIN {X 0,Y 594.539,Z 632.95,A -85,B 0,C 180,E1 -1184.231,E2 -1184.231} C_VEL
LIN {X 0,Y 594.678,Z 621.144,A -85,B 0,C 180,E1 -1185.333,E2 -1185.333} C_VEL
LIN {X 0,Y 594.809,Z 607.884,A -85,B 0,C 180,E1 -1186.385,E2 -1186.385} C_VEL
LIN {X 0,Y 594.95,Z 593.436,A -85,B 0,C 180,E1 -1187.354,E2 -1187.354} C_VEL
LIN {X 0,Y 595.045,Z 579.269,A -85,B 0,C 180,E1 -1188.15,E2 -1188.15} C_VEL
LIN {X 0,Y 595.199,Z 564.115,A -85,B 0,C 180,E1 -1188.854,E2 -1188.854} C_VEL
LIN {X 0,Y 595.279,Z 548.349,A -85,B 0,C 180,E1 -1189.438,E2 -1189.438} C_VEL
LIN {X 0,Y 595.386,Z 532.356,A -85,B 0,C 180,E1 -1189.883,E2 -1189.883} C_VEL
LIN {X 0,Y 595.461,Z 516.443,A -85,B 0,C 180,E1 -1190.195,E2 -1190.195} C_VEL
LIN {X 0,Y 595.784,Z 315.478,A -85,B 0,C 180,E1 -1192.748,E2 -1192.748} C_VEL
LIN {X 0,Y 595.216,Z 312.031,A -85,B 0,C 180,E1 -1192.816,E2 -1192.816} C_VEL
LIN {X 0,Y 595.477,Z 276.405,A -85,B 0,C 180,E1 -1195.798,E2 -1195.798} C_VEL
LIN {X 0,Y 595.55,Z 265.363,A -85,B 0,C 180,E1 -1196.738,E2 -1196.738} C_VEL
LIN {X 0,Y 594.394,Z 260.761,A -85,B 0,C 180,E1 -1197.198,E2 -1197.198} C_VEL
LIN {X 0,Y 594.372,Z 260.759,A -85,B 0,C 180,E1 -1199.776,E2 -1199.776} C_VEL
LIN {X 0,Y 594.357,Z 260.757,A -85,B 0,C 180,E1 -1202.147,E2 -1202.147} C_VEL
LIN {X 0,Y 594.371,Z 260.755,A -85,B 0,C 180,E1 -1204.58,E2 -1204.58} C_VEL
LIN {X 0,Y 594.387,Z 260.758,A -85,B 0,C 180,E1 -1207.608,E2 -1207.608} C_VEL
LIN {X 0,Y 594.363,Z 260.756,A -85,B 0,C 180,E1 -1210.567,E2 -1210.567} C_VEL
LIN {X 0,Y 594.376,Z 260.764,A -85,B 0,C 180,E1 -1213.298,E2 -1213.298} C_VEL
LIN {X 0,Y 594.364,Z 260.755,A -85,B 0,C 180,E1 -1216.16,E2 -1216.16} C_VEL
LIN {X 0,Y 594.381,Z 260.762,A -85,B 0,C 180,E1 -1219.177,E2 -1219.177} C_VEL
LIN {X 0,Y 594.384,Z 260.752,A -85,B 0,C 180,E1 -1222.059,E2 -1222.059} C_VEL
LIN {X 0,Y 594.355,Z 260.758,A -85,B 0,C 180,E1 -1224.675,E2 -1224.675} C_VEL
LIN {X 0,Y 594.375,Z 260.762,A -85,B 0,C 180,E1 -1227.089,E2 -1227.089} C_VEL
LIN {X 0,Y 594.383,Z 260.755,A -85,B 0,C 180,E1 -1229.672,E2 -1229.672} C_VEL
LIN {X 0,Y 594.371,Z 260.755,A -85,B 0,C 180,E1 -1232.539,E2 -1232.539} C_VEL
LIN {X 0,Y 594.37,Z 260.759,A -85,B 0,C 180,E1 -1234.807,E2 -1234.807} C_VEL
LIN {X 0,Y 594.362,Z 260.764,A -85,B 0,C 180,E1 -1237.265,E2 -1237.265} C_VEL
LIN {X 0,Y 594.372,Z 260.752,A -85,B 0,C 180,E1 -1239.946,E2 -1239.946} C_VEL
LIN {X 0,Y 594.386,Z 260.757,A -85,B 0,C 180,E1 -1242.807,E2 -1242.807} C_VEL
LIN {X 0,Y 594.387,Z 260.751,A -85,B 0,C 180,E1 -1245.826,E2 -1245.826} C_VEL
LIN {X 0,Y 594.391,Z 260.752,A -85,B 0,C 180,E1 -1248.404,E2 -1248.404} C_VEL
LIN {X 0,Y 594.377,Z 260.762,A -85,B 0,C 180,E1 -1251.158,E2 -1251.158} C_VEL
LIN {X 0,Y 594.389,Z 260.75,A -85,B 0,C 180,E1 -1253.891,E2 -1253.891} C_VEL
LIN {X 0,Y 594.376,Z 260.757,A -85,B 0,C 180,E1 -1256.611,E2 -1256.611} C_VEL
LIN {X 0,Y 594.419,Z 260.752,A -85,B 0,C 180,E1 -1259.323,E2 -1259.323} C_VEL
LIN {X 0,Y 594.403,Z 260.749,A -85,B 0,C 180,E1 -1262.033,E2 -1262.033} C_VEL
LIN {X 0,Y 594.386,Z 260.758,A -85,B 0,C 180,E1 -1264.748,E2 -1264.748} C_VEL
LIN {X 0,Y 594.393,Z 260.752,A -85,B 0,C 180,E1 -1267.473,E2 -1267.473} C_VEL
LIN {X 0,Y 594.391,Z 260.751,A -85,B 0,C 180,E1 -1270.216,E2 -1270.216} C_VEL
LIN {X 0,Y 594.364,Z 260.765,A -85,B 0,C 180,E1 -1272.983,E2 -1272.983} C_VEL
LIN {X 0,Y 594.358,Z 260.759,A -85,B 0,C 180,E1 -1275.321,E2 -1275.321} C_VEL
LIN {X 0,Y 593.685,Z 260.84,A -85,B 0,C 180,E1 -1275.887,E2 -1275.887} C_VEL
LIN {X 0,Y 590.82,Z 261.202,A -85,B 0,C 180,E1 -1276.805,E2 -1276.805} C_VEL
LIN {X 0,Y 588.411,Z 261.499,A -85,B 0,C 180,E1 -1277.544,E2 -1277.544} C_VEL
LIN {X 0,Y 587.387,Z 261.624,A -85,B 0,C 180,E1 -1278.114,E2 -1278.114} C_VEL
LIN {X 0,Y 587.309,Z 261.635,A -85,B 0,C 180,E1 -1278.307,E2 -1278.307} C_VEL
LIN {X 0,Y 587.328,Z 261.638,A -85,B 0,C 180,E1 -1281.038,E2 -1281.038} C_VEL
LIN {X 0,Y 587.321,Z 261.637,A -85,B 0,C 180,E1 -1283.259,E2 -1283.259} C_VEL
LIN {X 0,Y 587.329,Z 261.633,A -85,B 0,C 180,E1 -1285.517,E2 -1285.517} C_VEL
LIN {X 0,Y 587.345,Z 261.627,A -85,B 0,C 180,E1 -1287.818,E2 -1287.818} C_VEL
LIN {X 0,Y 587.335,Z 261.635,A -85,B 0,C 180,E1 -1290.51,E2 -1290.51} C_VEL
LIN {X 0,Y 587.331,Z 261.633,A -85,B 0,C 180,E1 -1293.397,E2 -1293.397} C_VEL
LIN {X 0,Y 587.354,Z 261.628,A -85,B 0,C 180,E1 -1295.896,E2 -1295.896} C_VEL
LIN {X 0,Y 587.329,Z 261.634,A -85,B 0,C 180,E1 -1298.479,E2 -1298.479} C_VEL
LIN {X 0,Y 587.334,Z 261.635,A -85,B 0,C 180,E1 -1301.157,E2 -1301.157} C_VEL
LIN {X 0,Y 587.325,Z 261.633,A -85,B 0,C 180,E1 -1304.114,E2 -1304.114} C_VEL
LIN {X 0,Y 587.319,Z 261.64,A -85,B 0,C 180,E1 -1306.994,E2 -1306.994} C_VEL
LIN {X 0,Y 587.316,Z 261.633,A -85,B 0,C 180,E1 -1309.746,E2 -1309.746} C_VEL
LIN {X 0,Y 587.344,Z 261.633,A -85,B 0,C 180,E1 -1312.393,E2 -1312.393} C_VEL
LIN {X 0,Y 587.357,Z 261.628,A -85,B 0,C 180,E1 -1315.78,E2 -1315.78} C_VEL
LIN {X 0,Y 587.343,Z 261.632,A -85,B 0,C 180,E1 -1318.231,E2 -1318.231} C_VEL
LIN {X 0,Y 587.345,Z 261.639,A -85,B 0,C 180,E1 -1320.868,E2 -1320.868} C_VEL
LIN {X 0,Y 587.358,Z 261.63,A -85,B 0,C 180,E1 -1323.819,E2 -1323.819} C_VEL
LIN {X 0,Y 587.368,Z 261.762,A -85,B 0,C 180,E1 -1324.878,E2 -1324.878} C_VEL
LIN {X 0,Y 588.472,Z 266.97,A -85,B 0,C 180,E1 -1325.433,E2 -1325.433} C_VEL
LIN {X 0,Y 588.319,Z 282.8,A -85,B 0,C 180,E1 -1326.949,E2 -1326.949} C_VEL
LIN {X 0,Y 589.23,Z 287.887,A -85,B 0,C 180,E1 -1327.061,E2 -1327.061} C_VEL
LIN {X 0,Y 588.802,Z 487.987,A -85,B 0,C 180,E1 -1329.634,E2 -1329.634} C_VEL
LIN {X 0,Y 588.706,Z 504.205,A -85,B 0,C 180,E1 -1329.973,E2 -1329.973} C_VEL
LIN {X 0,Y 588.559,Z 520.958,A -85,B 0,C 180,E1 -1330.467,E2 -1330.467} C_VEL
LIN {X 0,Y 588.402,Z 536.858,A -85,B 0,C 180,E1 -1331.084,E2 -1331.084} C_VEL
LIN {X 0,Y 588.247,Z 551.894,A -85,B 0,C 180,E1 -1331.813,E2 -1331.813} C_VEL
LIN {X 0,Y 588.028,Z 567.628,A -85,B 0,C 180,E1 -1332.747,E2 -1332.747} C_VEL
LIN {X 0,Y 587.894,Z 580.793,A -85,B 0,C 180,E1 -1333.684,E2 -1333.684} C_VEL
LIN {X 0,Y 587.679,Z 593.58,A -85,B 0,C 180,E1 -1334.746,E2 -1334.746} C_VEL
LIN {X 0,Y 587.57,Z 606.208,A -85,B 0,C 180,E1 -1335.982,E2 -1335.982} C_VEL
LIN {X 0,Y 587.427,Z 616.986,A -85,B 0,C 180,E1 -1337.213,E2 -1337.213} C_VEL
LIN {X 0,Y 587.362,Z 627.363,A -85,B 0,C 180,E1 -1338.614,E2 -1338.614} C_VEL
LIN {X 0,Y 587.279,Z 636.025,A -85,B 0,C 180,E1 -1340.007,E2 -1340.007} C_VEL
LIN {X 0,Y 587.239,Z 643.278,A -85,B 0,C 180,E1 -1341.396,E2 -1341.396} C_VEL
LIN {X 0,Y 587.21,Z 649.288,A -85,B 0,C 180,E1 -1342.781,E2 -1342.781} C_VEL
LIN {X 0,Y 587.188,Z 655.109,A -85,B 0,C 180,E1 -1344.505,E2 -1344.505} C_VEL
LIN {X 0,Y 587.17,Z 658.54,A -85,B 0,C 180,E1 -1345.882,E2 -1345.882} C_VEL
LIN {X 0,Y 587.12,Z 661.016,A -85,B 0,C 180,E1 -1347.256,E2 -1347.256} C_VEL
LIN {X 0,Y 587.142,Z 662.448,A -85,B 0,C 180,E1 -1348.628,E2 -1348.628} C_VEL
LIN {X 0,Y 587.133,Z 662.996,A -85,B 0,C 180,E1 -1350,E2 -1350} C_VEL
LIN {X 0,Y 587.139,Z 662.509,A -85,B 0,C 180,E1 -1351.372,E2 -1351.372} C_VEL
LIN {X 0,Y 587.12,Z 661.151,A -85,B 0,C 180,E1 -1352.744,E2 -1352.744} C_VEL
LIN {X 0,Y 587.167,Z 658.729,A -85,B 0,C 180,E1 -1354.118,E2 -1354.118} C_VEL
LIN {X 0,Y 587.189,Z 655.382,A -85,B 0,C 180,E1 -1355.494,E2 -1355.494} C_VEL
LIN {X 0,Y 587.21,Z 649.638,A -85,B 0,C 180,E1 -1357.219,E2 -1357.219} C_VEL
LIN {X 0,Y 587.239,Z 643.698,A -85,B 0,C 180,E1 -1358.604,E2 -1358.604} C_VEL
LIN {X 0,Y 587.291,Z 635.536,A -85,B 0,C 180,E1 -1360.166,E2 -1360.166} C_VEL
LIN {X 0,Y 587.351,Z 626.765,A -85,B 0,C 180,E1 -1361.561,E2 -1361.561} C_VEL
LIN {X 0,Y 587.447,Z 616.29,A -85,B 0,C 180,E1 -1362.963,E2 -1362.963} C_VEL
LIN {X 0,Y 587.563,Z 605.353,A -85,B 0,C 180,E1 -1364.201,E2 -1364.201} C_VEL
LIN {X 0,Y 587.676,Z 594.564,A -85,B 0,C 180,E1 -1365.254,E2 -1365.254} C_VEL
LIN {X 0,Y 587.837,Z 580.803,A -85,B 0,C 180,E1 -1366.406,E2 -1366.406} C_VEL
LIN {X 0,Y 588.044,Z 566.97,A -85,B 0,C 180,E1 -1367.385,E2 -1367.385} C_VEL
LIN {X 0,Y 588.237,Z 551.896,A -85,B 0,C 180,E1 -1368.278,E2 -1368.278} C_VEL
LIN {X 0,Y 588.431,Z 536.593,A -85,B 0,C 180,E1 -1369.017,E2 -1369.017} C_VEL
LIN {X 0,Y 588.543,Z 520.938,A -85,B 0,C 180,E1 -1369.624,E2 -1369.624} C_VEL
LIN {X 0,Y 588.726,Z 504.163,A -85,B 0,C 180,E1 -1370.118,E2 -1370.118} C_VEL
LIN {X 0,Y 588.81,Z 487.911,A -85,B 0,C 180,E1 -1370.456,E2 -1370.456} C_VEL
LIN {X 0,Y 589.205,Z 287.145,A -85,B 0,C 180,E1 -1373.04,E2 -1373.04} C_VEL
LIN {X 0,Y 588.321,Z 282.631,A -85,B 0,C 180,E1 -1373.157,E2 -1373.157} C_VEL
LIN {X 0,Y 588.341,Z 265.658,A -85,B 0,C 180,E1 -1374.79,E2 -1374.79} C_VEL
LIN {X 0,Y 587.334,Z 261.64,A -85,B 0,C 180,E1 -1375.232,E2 -1375.232} C_VEL
LIN {X 0,Y 587.337,Z 261.635,A -85,B 0,C 180,E1 -1377.818,E2 -1377.818} C_VEL
LIN {X 0,Y 587.334,Z 261.632,A -85,B 0,C 180,E1 -1380.509,E2 -1380.509} C_VEL
LIN {X 0,Y 587.334,Z 261.641,A -85,B 0,C 180,E1 -1383.396,E2 -1383.396} C_VEL
LIN {X 0,Y 587.289,Z 261.637,A -85,B 0,C 180,E1 -1385.9,E2 -1385.9} C_VEL
LIN {X 0,Y 587.321,Z 261.633,A -85,B 0,C 180,E1 -1388.48,E2 -1388.48} C_VEL
LIN {X 0,Y 587.334,Z 261.639,A -85,B 0,C 180,E1 -1391.157,E2 -1391.157} C_VEL
LIN {X 0,Y 587.333,Z 261.631,A -85,B 0,C 180,E1 -1394.114,E2 -1394.114} C_VEL
LIN {X 0,Y 587.311,Z 261.639,A -85,B 0,C 180,E1 -1396.993,E2 -1396.993} C_VEL
LIN {X 0,Y 587.312,Z 261.636,A -85,B 0,C 180,E1 -1399.745,E2 -1399.745} C_VEL
LIN {X 0,Y 587.342,Z 261.63,A -85,B 0,C 180,E1 -1402.392,E2 -1402.392} C_VEL
LIN {X 0,Y 587.329,Z 261.637,A -85,B 0,C 180,E1 -1404.944,E2 -1404.944} C_VEL
LIN {X 0,Y 587.335,Z 261.636,A -85,B 0,C 180,E1 -1407.421,E2 -1407.421} C_VEL
LIN {X 0,Y 587.331,Z 261.632,A -85,B 0,C 180,E1 -1409.83,E2 -1409.83} C_VEL
LIN {X 0,Y 587.349,Z 261.627,A -85,B 0,C 180,E1 -1412.307,E2 -1412.307} C_VEL
LIN {X 0,Y 587.348,Z 261.637,A -85,B 0,C 180,E1 -1415.241,E2 -1415.241} C_VEL
LIN {X 0,Y 587.319,Z 261.631,A -85,B 0,C 180,E1 -1418.226,E2 -1418.226} C_VEL
LIN {X 0,Y 587.347,Z 261.639,A -85,B 0,C 180,E1 -1421.151,E2 -1421.151} C_VEL
LIN {X 0,Y 587.321,Z 261.63,A -85,B 0,C 180,E1 -1424.025,E2 -1424.025} C_VEL
LIN {X 0,Y 587.357,Z 261.628,A -85,B 0,C 180,E1 -1426.154,E2 -1426.154} C_VEL
LIN {X 0,Y 587.34,Z 261.639,A -85,B 0,C 180,E1 -1428.962,E2 -1428.962} C_VEL
LIN {X 0,Y 587.363,Z 261.627,A -85,B 0,C 180,E1 -1431.745,E2 -1431.745} C_VEL
LIN {X 0,Y 587.361,Z 261.63,A -85,B 0,C 180,E1 -1434.507,E2 -1434.507} C_VEL
LIN {X 0,Y 587.369,Z 261.631,A -85,B 0,C 180,E1 -1437.257,E2 -1437.257} C_VEL
LIN {X 0,Y 587.382,Z 261.625,A -85,B 0,C 180,E1 -1440,E2 -1440} C_VEL
LIN {X 0,Y 587.369,Z 261.632,A -85,B 0,C 180,E1 -1442.743,E2 -1442.743} C_VEL
LIN {X 0,Y 587.361,Z 261.629,A -85,B 0,C 180,E1 -1445.493,E2 -1445.493} C_VEL
LIN {X 0,Y 587.363,Z 261.628,A -85,B 0,C 180,E1 -1448.255,E2 -1448.255} C_VEL
LIN {X 0,Y 587.345,Z 261.636,A -85,B 0,C 180,E1 -1451.134,E2 -1451.134} C_VEL
LIN {X 0,Y 587.362,Z 261.628,A -85,B 0,C 180,E1 -1454.261,E2 -1454.261} C_VEL
LIN {X 0,Y 587.347,Z 261.632,A -85,B 0,C 180,E1 -1457.406,E2 -1457.406} C_VEL
LIN {X 0,Y 587.327,Z 261.634,A -85,B 0,C 180,E1 -1460.305,E2 -1460.305} C_VEL
LIN {X 0,Y 587.32,Z 261.637,A -85,B 0,C 180,E1 -1463.259,E2 -1463.259} C_VEL
LIN {X 0,Y 587.328,Z 261.633,A -85,B 0,C 180,E1 -1465.517,E2 -1465.517} C_VEL
LIN {X 0,Y 587.344,Z 261.63,A -85,B 0,C 180,E1 -1467.818,E2 -1467.818} C_VEL
LIN {X 0,Y 587.334,Z 261.636,A -85,B 0,C 180,E1 -1470.51,E2 -1470.51} C_VEL
LIN {X 0,Y 587.33,Z 261.634,A -85,B 0,C 180,E1 -1473.397,E2 -1473.397} C_VEL
LIN {X 0,Y 587.353,Z 261.629,A -85,B 0,C 180,E1 -1475.895,E2 -1475.895} C_VEL
LIN {X 0,Y 587.327,Z 261.637,A -85,B 0,C 180,E1 -1478.479,E2 -1478.479} C_VEL
LIN {X 0,Y 587.334,Z 261.635,A -85,B 0,C 180,E1 -1481.157,E2 -1481.157} C_VEL
LIN {X 0,Y 587.323,Z 261.634,A -85,B 0,C 180,E1 -1484.113,E2 -1484.113} C_VEL
LIN {X 0,Y 587.316,Z 261.639,A -85,B 0,C 180,E1 -1486.994,E2 -1486.994} C_VEL
LIN {X 0,Y 587.314,Z 261.634,A -85,B 0,C 180,E1 -1489.746,E2 -1489.746} C_VEL
LIN {X 0,Y 587.342,Z 261.635,A -85,B 0,C 180,E1 -1492.392,E2 -1492.392} C_VEL
LIN {X 0,Y 587.342,Z 261.628,A -85,B 0,C 180,E1 -1495.653,E2 -1495.653} C_VEL
LIN {X 0,Y 587.341,Z 261.634,A -85,B 0,C 180,E1 -1498.231,E2 -1498.231} C_VEL
LIN {X 0,Y 587.343,Z 261.639,A -85,B 0,C 180,E1 -1500.868,E2 -1500.868} C_VEL
LIN {X 0,Y 587.361,Z 261.804,A -85,B 0,C 180,E1 -1502.548,E2 -1502.548} C_VEL
LIN {X 0,Y 588.685,Z 266.468,A -85,B 0,C 180,E1 -1503.021,E2 -1503.021} C_VEL
LIN {X 0,Y 588.858,Z 273.996,A -85,B 0,C 180,E1 -1503.682,E2 -1503.682} C_VEL
LIN {X 0,Y 588.507,Z 309.53,A -85,B 0,C 180,E1 -1506.698,E2 -1506.698} C_VEL
LIN {X 0,Y 588.488,Z 311.98,A -85,B 0,C 180,E1 -1506.904,E2 -1506.904} C_VEL
LIN {X 0,Y 589.247,Z 317.687,A -85,B 0,C 180,E1 -1507.014,E2 -1507.014} C_VEL
LIN {X 0,Y 588.805,Z 517.95,A -85,B 0,C 180,E1 -1509.589,E2 -1509.589} C_VEL
LIN {X 0,Y 588.706,Z 534.184,A -85,B 0,C 180,E1 -1509.927,E2 -1509.927} C_VEL
LIN {X 0,Y 588.547,Z 550.95,A -85,B 0,C 180,E1 -1510.421,E2 -1510.421} C_VEL
LIN {X 0,Y 588.406,Z 566.726,A -85,B 0,C 180,E1 -1511.033,E2 -1511.033} C_VEL
LIN {X 0,Y 588.248,Z 581.023,A -85,B 0,C 180,E1 -1511.723,E2 -1511.723} C_VEL
LIN {X 0,Y 588.076,Z 594.851,A -85,B 0,C 180,E1 -1512.527,E2 -1512.527} C_VEL
LIN {X 0,Y 587.916,Z 609.055,A -85,B 0,C 180,E1 -1513.506,E2 -1513.506} C_VEL
LIN {X 0,Y 587.729,Z 622.125,A -85,B 0,C 180,E1 -1514.57,E2 -1514.57} C_VEL
LIN {X 0,Y 587.563,Z 633.628,A -85,B 0,C 180,E1 -1515.664,E2 -1515.664} C_VEL
LIN {X 0,Y 587.449,Z 644.425,A -85,B 0,C 180,E1 -1516.861,E2 -1516.861} C_VEL
LIN {X 0,Y 587.351,Z 655.21,A -85,B 0,C 180,E1 -1518.263,E2 -1518.263} C_VEL
LIN {X 0,Y 587.297,Z 664.262,A -85,B 0,C 180,E1 -1519.659,E2 -1519.659} C_VEL
LIN {X 0,Y 587.245,Z 671.857,A -85,B 0,C 180,E1 -1521.05,E2 -1521.05} C_VEL
LIN {X 0,Y 587.207,Z 679.468,A -85,B 0,C 180,E1 -1522.781,E2 -1522.781} C_VEL
LIN {X 0,Y 587.187,Z 685.247,A -85,B 0,C 180,E1 -1524.506,E2 -1524.506} C_VEL
LIN {X 0,Y 587.168,Z 688.635,A -85,B 0,C 180,E1 -1525.882,E2 -1525.882} C_VEL
LIN {X 0,Y 587.119,Z 691.088,A -85,B 0,C 180,E1 -1527.256,E2 -1527.256} C_VEL
LIN {X 0,Y 587.14,Z 692.478,A -85,B 0,C 180,E1 -1528.628,E2 -1528.628} C_VEL
LIN {X 0,Y 587.132,Z 693,A -85,B 0,C 180,E1 -1530,E2 -1530} C_VEL
LIN {X 0,Y 587.14,Z 692.478,A -85,B 0,C 180,E1 -1531.372,E2 -1531.372} C_VEL
LIN {X 0,Y 587.119,Z 691.087,A -85,B 0,C 180,E1 -1532.744,E2 -1532.744} C_VEL
LIN {X 0,Y 587.168,Z 688.634,A -85,B 0,C 180,E1 -1534.118,E2 -1534.118} C_VEL
LIN {X 0,Y 587.187,Z 684.186,A -85,B 0,C 180,E1 -1535.839,E2 -1535.839} C_VEL
LIN {X 0,Y 587.207,Z 679.468,A -85,B 0,C 180,E1 -1537.219,E2 -1537.219} C_VEL
LIN {X 0,Y 587.245,Z 671.857,A -85,B 0,C 180,E1 -1538.95,E2 -1538.95} C_VEL
LIN {X 0,Y 587.302,Z 663.249,A -85,B 0,C 180,E1 -1540.515,E2 -1540.515} C_VEL
LIN {X 0,Y 587.366,Z 653.972,A -85,B 0,C 180,E1 -1541.911,E2 -1541.911} C_VEL
LIN {X 0,Y 587.449,Z 644.424,A -85,B 0,C 180,E1 -1543.139,E2 -1543.139} C_VEL
LIN {X 0,Y 587.589,Z 632.57,A -85,B 0,C 180,E1 -1544.441,E2 -1544.441} C_VEL
LIN {X 0,Y 587.759,Z 620.097,A -85,B 0,C 180,E1 -1545.607,E2 -1545.607} C_VEL
LIN {X 0,Y 587.909,Z 606.708,A -85,B 0,C 180,E1 -1546.672,E2 -1546.672} C_VEL
LIN {X 0,Y 588.118,Z 592.009,A -85,B 0,C 180,E1 -1547.652,E2 -1547.652} C_VEL
LIN {X 0,Y 588.288,Z 577.524,A -85,B 0,C 180,E1 -1548.456,E2 -1548.456} C_VEL
LIN {X 0,Y 588.444,Z 562.396,A -85,B 0,C 180,E1 -1549.149,E2 -1549.149} C_VEL
LIN {X 0,Y 588.617,Z 546.253,A -85,B 0,C 180,E1 -1549.735,E2 -1549.735} C_VEL
LIN {X 0,Y 588.753,Z 529.608,A -85,B 0,C 180,E1 -1550.185,E2 -1550.185} C_VEL
LIN {X 0,Y 588.796,Z 513.43,A -85,B 0,C 180,E1 -1550.48,E2 -1550.48} C_VEL
LIN {X 0,Y 589.249,Z 316.703,A -85,B 0,C 180,E1 -1552.999,E2 -1552.999} C_VEL
LIN {X 0,Y 588.478,Z 312.01,A -85,B 0,C 180,E1 -1553.094,E2 -1553.094} C_VEL
LIN {X 0,Y 588.827,Z 276.405,A -85,B 0,C 180,E1 -1556.112,E2 -1556.112} C_VEL
LIN {X 0,Y 588.898,Z 268.349,A -85,B 0,C 180,E1 -1556.805,E2 -1556.805} C_VEL
LIN {X 0,Y 588.069,Z 264.275,A -85,B 0,C 180,E1 -1557.2,E2 -1557.2} C_VEL
LIN {X 0,Y 587.341,Z 261.64,A -85,B 0,C 180,E1 -1557.477,E2 -1557.477} C_VEL
LIN {X 0,Y 587.33,Z 261.633,A -85,B 0,C 180,E1 -1560.17,E2 -1560.17} C_VEL
LIN {X 0,Y 587.332,Z 261.633,A -85,B 0,C 180,E1 -1562.579,E2 -1562.579} C_VEL
LIN {X 0,Y 587.32,Z 261.639,A -85,B 0,C 180,E1 -1565.056,E2 -1565.056} C_VEL
LIN {X 0,Y 587.338,Z 261.633,A -85,B 0,C 180,E1 -1567.839,E2 -1567.839} C_VEL
LIN {X 0,Y 587.313,Z 261.634,A -85,B 0,C 180,E1 -1570.254,E2 -1570.254} C_VEL
LIN {X 0,Y 587.316,Z 261.639,A -85,B 0,C 180,E1 -1573.006,E2 -1573.006} C_VEL
LIN {X 0,Y 587.323,Z 261.633,A -85,B 0,C 180,E1 -1575.887,E2 -1575.887} C_VEL
LIN {X 0,Y 587.334,Z 261.634,A -85,B 0,C 180,E1 -1578.843,E2 -1578.843} C_VEL
LIN {X 0,Y 587.327,Z 261.637,A -85,B 0,C 180,E1 -1581.521,E2 -1581.521} C_VEL
LIN {X 0,Y 587.317,Z 261.633,A -85,B 0,C 180,E1 -1584.102,E2 -1584.102} C_VEL
LIN {X 0,Y 587.33,Z 261.633,A -85,B 0,C 180,E1 -1586.603,E2 -1586.603} C_VEL
LIN {X 0,Y 587.334,Z 261.636,A -85,B 0,C 180,E1 -1589.49,E2 -1589.49} C_VEL
LIN {X 0,Y 587.348,Z 261.629,A -85,B 0,C 180,E1 -1592.307,E2 -1592.307} C_VEL
LIN {X 0,Y 587.348,Z 261.638,A -85,B 0,C 180,E1 -1595.241,E2 -1595.241} C_VEL
LIN {X 0,Y 587.318,Z 261.632,A -85,B 0,C 180,E1 -1598.226,E2 -1598.226} C_VEL
LIN {X 0,Y 587.347,Z 261.638,A -85,B 0,C 180,E1 -1601.151,E2 -1601.151} C_VEL
LIN {X 0,Y 587.321,Z 261.632,A -85,B 0,C 180,E1 -1604.025,E2 -1604.025} C_VEL
LIN {X 0,Y 587.357,Z 261.625,A -85,B 0,C 180,E1 -1606.154,E2 -1606.154} C_VEL
LIN {X 0,Y 587.341,Z 261.637,A -85,B 0,C 180,E1 -1608.963,E2 -1608.963} C_VEL
LIN {X 0,Y 587.363,Z 261.627,A -85,B 0,C 180,E1 -1611.745,E2 -1611.745} C_VEL
LIN {X 0,Y 587.359,Z 261.627,A -85,B 0,C 180,E1 -1614.507,E2 -1614.507} C_VEL
LIN {X 0,Y 587.37,Z 261.633,A -85,B 0,C 180,E1 -1617.257,E2 -1617.257} C_VEL
LIN {X 0,Y 587.382,Z 261.623,A -85,B 0,C 180,E1 -1620,E2 -1620} C_VEL
LIN {X 0,Y 587.368,Z 261.63,A -85,B 0,C 180,E1 -1622.743,E2 -1622.743} C_VEL
LIN {X 0,Y 587.361,Z 261.63,A -85,B 0,C 180,E1 -1625.493,E2 -1625.493} C_VEL
LIN {X 0,Y 587.364,Z 261.625,A -85,B 0,C 180,E1 -1628.255,E2 -1628.255} C_VEL
LIN {X 0,Y 587.346,Z 261.637,A -85,B 0,C 180,E1 -1631.134,E2 -1631.134} C_VEL
LIN {X 0,Y 587.363,Z 261.627,A -85,B 0,C 180,E1 -1634.261,E2 -1634.261} C_VEL
LIN {X 0,Y 587.348,Z 261.632,A -85,B 0,C 180,E1 -1637.406,E2 -1637.406} C_VEL
LIN {X 0,Y 587.309,Z 261.635,A -85,B 0,C 180,E1 -1638.307,E2 -1638.307} C_VEL
LIN {X 0,Y 586.664,Z 261.723,A -85,B 0,C 180,E1 -1638.879,E2 -1638.879} C_VEL
LIN {X 0,Y 583.839,Z 262.076,A -85,B 0,C 180,E1 -1639.808,E2 -1639.808} C_VEL
LIN {X 0,Y 581.429,Z 262.374,A -85,B 0,C 180,E1 -1640.555,E2 -1640.555} C_VEL
LIN {X 0,Y 580.376,Z 262.502,A -85,B 0,C 180,E1 -1641.131,E2 -1641.131} C_VEL
LIN {X 0,Y 580.281,Z 262.51,A -85,B 0,C 180,E1 -1641.326,E2 -1641.326} C_VEL
LIN {X 0,Y 580.278,Z 262.511,A -85,B 0,C 180,E1 -1643.558,E2 -1643.558} C_VEL
LIN {X 0,Y 580.288,Z 262.508,A -85,B 0,C 180,E1 -1645.849,E2 -1645.849} C_VEL
LIN {X 0,Y 580.297,Z 262.505,A -85,B 0,C 180,E1 -1648.186,E2 -1648.186} C_VEL
LIN {X 0,Y 580.283,Z 262.516,A -85,B 0,C 180,E1 -1650.695,E2 -1650.695} C_VEL
LIN {X 0,Y 580.3,Z 262.51,A -85,B 0,C 180,E1 -1653.316,E2 -1653.316} C_VEL
LIN {X 0,Y 580.324,Z 262.504,A -85,B 0,C 180,E1 -1655.768,E2 -1655.768} C_VEL
LIN {X 0,Y 580.287,Z 262.507,A -85,B 0,C 180,E1 -1658.146,E2 -1658.146} C_VEL
LIN {X 0,Y 580.297,Z 262.517,A -85,B 0,C 180,E1 -1660.844,E2 -1660.844} C_VEL
LIN {X 0,Y 580.277,Z 262.51,A -85,B 0,C 180,E1 -1663.658,E2 -1663.658} C_VEL
LIN {X 0,Y 580.284,Z 262.514,A -85,B 0,C 180,E1 -1666.609,E2 -1666.609} C_VEL
LIN {X 0,Y 580.298,Z 262.512,A -85,B 0,C 180,E1 -1669.157,E2 -1669.157} C_VEL
LIN {X 0,Y 580.289,Z 262.508,A -85,B 0,C 180,E1 -1671.927,E2 -1671.927} C_VEL
LIN {X 0,Y 580.25,Z 262.518,A -85,B 0,C 180,E1 -1674.453,E2 -1674.453} C_VEL
LIN {X 0,Y 580.289,Z 262.515,A -85,B 0,C 180,E1 -1676.975,E2 -1676.975} C_VEL
LIN {X 0,Y 580.298,Z 262.51,A -85,B 0,C 180,E1 -1679.425,E2 -1679.425} C_VEL
LIN {X 0,Y 580.295,Z 262.511,A -85,B 0,C 180,E1 -1682.142,E2 -1682.142} C_VEL
LIN {X 0,Y 580.314,Z 262.603,A -85,B 0,C 180,E1 -1684.633,E2 -1684.633} C_VEL
LIN {X 0,Y 581.695,Z 268.354,A -85,B 0,C 180,E1 -1685.263,E2 -1685.263} C_VEL
LIN {X 0,Y 581.551,Z 282.892,A -85,B 0,C 180,E1 -1686.674,E2 -1686.674} C_VEL
LIN {X 0,Y 582.713,Z 288.647,A -85,B 0,C 180,E1 -1686.799,E2 -1686.799} C_VEL
LIN {X 0,Y 582.146,Z 488.025,A -85,B 0,C 180,E1 -1689.391,E2 -1689.391} C_VEL
LIN {X 0,Y 582.021,Z 504.23,A -85,B 0,C 180,E1 -1689.732,E2 -1689.732} C_VEL
LIN {X 0,Y 581.835,Z 520.974,A -85,B 0,C 180,E1 -1690.232,E2 -1690.232} C_VEL
LIN {X 0,Y 581.656,Z 537.023,A -85,B 0,C 180,E1 -1690.863,E2 -1690.863} C_VEL
LIN {X 0,Y 581.443,Z 551.907,A -85,B 0,C 180,E1 -1691.592,E2 -1691.592} C_VEL
LIN {X 0,Y 581.199,Z 566.707,A -85,B 0,C 180,E1 -1692.477,E2 -1692.477} C_VEL
LIN {X 0,Y 581.004,Z 580.803,A -85,B 0,C 180,E1 -1693.485,E2 -1693.485} C_VEL
LIN {X 0,Y 580.744,Z 593.584,A -85,B 0,C 180,E1 -1694.56,E2 -1694.56} C_VEL
LIN {X 0,Y 580.616,Z 605.2,A -85,B 0,C 180,E1 -1695.699,E2 -1695.699} C_VEL
LIN {X 0,Y 580.413,Z 616.991,A -85,B 0,C 180,E1 -1697.055,E2 -1697.055} C_VEL
LIN {X 0,Y 580.323,Z 627.366,A -85,B 0,C 180,E1 -1698.474,E2 -1698.474} C_VEL
LIN {X 0,Y 580.22,Z 636.028,A -85,B 0,C 180,E1 -1699.885,E2 -1699.885} C_VEL
LIN {X 0,Y 580.165,Z 643.281,A -85,B 0,C 180,E1 -1701.291,E2 -1701.291} C_VEL
LIN {X 0,Y 580.121,Z 649.29,A -85,B 0,C 180,E1 -1702.692,E2 -1702.692} C_VEL
LIN {X 0,Y 580.112,Z 655.111,A -85,B 0,C 180,E1 -1704.438,E2 -1704.438} C_VEL
LIN {X 0,Y 580.088,Z 658.542,A -85,B 0,C 180,E1 -1705.831,E2 -1705.831} C_VEL
LIN {X 0,Y 580.032,Z 661.017,A -85,B 0,C 180,E1 -1707.222,E2 -1707.222} C_VEL
LIN {X 0,Y 580.041,Z 662.448,A -85,B 0,C 180,E1 -1708.611,E2 -1708.611} C_VEL
LIN {X 0,Y 580.034,Z 662.996,A -85,B 0,C 180,E1 -1710,E2 -1710} C_VEL
LIN {X 0,Y 580.039,Z 662.509,A -85,B 0,C 180,E1 -1711.389,E2 -1711.389} C_VEL
LIN {X 0,Y 580.032,Z 661.151,A -85,B 0,C 180,E1 -1712.778,E2 -1712.778} C_VEL
LIN {X 0,Y 580.085,Z 658.728,A -85,B 0,C 180,E1 -1714.169,E2 -1714.169} C_VEL
LIN {X 0,Y 580.113,Z 655.381,A -85,B 0,C 180,E1 -1715.562,E2 -1715.562} C_VEL
LIN {X 0,Y 580.121,Z 649.636,A -85,B 0,C 180,E1 -1717.308,E2 -1717.308} C_VEL
LIN {X 0,Y 580.165,Z 643.696,A -85,B 0,C 180,E1 -1718.709,E2 -1718.709} C_VEL
LIN {X 0,Y 580.242,Z 635.534,A -85,B 0,C 180,E1 -1720.291,E2 -1720.291} C_VEL
LIN {X 0,Y 580.303,Z 626.759,A -85,B 0,C 180,E1 -1721.704,E2 -1721.704} C_VEL
LIN {X 0,Y 580.437,Z 616.285,A -85,B 0,C 180,E1 -1723.122,E2 -1723.122} C_VEL
LIN {X 0,Y 580.582,Z 604.758,A -85,B 0,C 180,E1 -1724.441,E2 -1724.441} C_VEL
LIN {X 0,Y 580.783,Z 592.611,A -85,B 0,C 180,E1 -1725.619,E2 -1725.619} C_VEL
LIN {X 0,Y 580.982,Z 579.636,A -85,B 0,C 180,E1 -1726.696,E2 -1726.696} C_VEL
LIN {X 0,Y 581.214,Z 565.553,A -85,B 0,C 180,E1 -1727.686,E2 -1727.686} C_VEL
LIN {X 0,Y 581.459,Z 551.888,A -85,B 0,C 180,E1 -1728.498,E2 -1728.498} C_VEL
LIN {X 0,Y 581.652,Z 536.936,A -85,B 0,C 180,E1 -1729.231,E2 -1729.231} C_VEL
LIN {X 0,Y 581.838,Z 520.92,A -85,B 0,C 180,E1 -1729.86,E2 -1729.86} C_VEL
LIN {X 0,Y 582.031,Z 504.141,A -85,B 0,C 180,E1 -1730.359,E2 -1730.359} C_VEL
LIN {X 0,Y 582.157,Z 487.872,A -85,B 0,C 180,E1 -1730.701,E2 -1730.701} C_VEL
LIN {X 0,Y 582.685,Z 288.325,A -85,B 0,C 180,E1 -1733.297,E2 -1733.297} C_VEL
LIN {X 0,Y 581.541,Z 282.823,A -85,B 0,C 180,E1 -1733.423,E2 -1733.423} C_VEL
LIN {X 0,Y 581.738,Z 268.874,A -85,B 0,C 180,E1 -1734.774,E2 -1734.774} C_VEL
LIN {X 0,Y 580.297,Z 262.518,A -85,B 0,C 180,E1 -1735.488,E2 -1735.488} C_VEL
LIN {X 0,Y 580.291,Z 262.511,A -85,B 0,C 180,E1 -1738.186,E2 -1738.186} C_VEL
LIN {X 0,Y 580.282,Z 262.512,A -85,B 0,C 180,E1 -1740.694,E2 -1740.694} C_VEL
LIN {X 0,Y 580.302,Z 262.515,A -85,B 0,C 180,E1 -1743.316,E2 -1743.316} C_VEL
LIN {X 0,Y 580.243,Z 262.515,A -85,B 0,C 180,E1 -1745.756,E2 -1745.756} C_VEL
LIN {X 0,Y 580.284,Z 262.51,A -85,B 0,C 180,E1 -1748.146,E2 -1748.146} C_VEL
LIN {X 0,Y 580.296,Z 262.511,A -85,B 0,C 180,E1 -1750.843,E2 -1750.843} C_VEL
LIN {X 0,Y 580.286,Z 262.513,A -85,B 0,C 180,E1 -1753.657,E2 -1753.657} C_VEL
LIN {X 0,Y 580.274,Z 262.511,A -85,B 0,C 180,E1 -1756.609,E2 -1756.609} C_VEL
LIN {X 0,Y 580.296,Z 262.516,A -85,B 0,C 180,E1 -1759.156,E2 -1759.156} C_VEL
LIN {X 0,Y 580.288,Z 262.509,A -85,B 0,C 180,E1 -1761.927,E2 -1761.927} C_VEL
LIN {X 0,Y 580.286,Z 262.509,A -85,B 0,C 180,E1 -1764.455,E2 -1764.455} C_VEL
LIN {X 0,Y 580.287,Z 262.515,A -85,B 0,C 180,E1 -1766.975,E2 -1766.975} C_VEL
LIN {X 0,Y 580.294,Z 262.514,A -85,B 0,C 180,E1 -1769.425,E2 -1769.425} C_VEL
LIN {X 0,Y 580.295,Z 262.505,A -85,B 0,C 180,E1 -1772.141,E2 -1772.141} C_VEL
LIN {X 0,Y 580.319,Z 262.512,A -85,B 0,C 180,E1 -1775.269,E2 -1775.269} C_VEL
LIN {X 0,Y 580.269,Z 262.508,A -85,B 0,C 180,E1 -1777.947,E2 -1777.947} C_VEL
LIN {X 0,Y 580.296,Z 262.514,A -85,B 0,C 180,E1 -1780.913,E2 -1780.913} C_VEL
LIN {X 0,Y 580.276,Z 262.508,A -85,B 0,C 180,E1 -1783.825,E2 -1783.825} C_VEL
LIN {X 0,Y 580.323,Z 262.504,A -85,B 0,C 180,E1 -1785.983,E2 -1785.983} C_VEL
LIN {X 0,Y 580.302,Z 262.513,A -85,B 0,C 180,E1 -1788.827,E2 -1788.827} C_VEL
LIN {X 0,Y 580.326,Z 262.505,A -85,B 0,C 180,E1 -1791.644,E2 -1791.644} C_VEL
LIN {X 0,Y 580.328,Z 262.505,A -85,B 0,C 180,E1 -1794.44,E2 -1794.44} C_VEL
LIN {X 0,Y 580.335,Z 262.507,A -85,B 0,C 180,E1 -1797.223,E2 -1797.223} C_VEL
LIN {X 0,Y 580.351,Z 262.5,A -85,B 0,C 180,E1 -1800,E2 -1800} C_VEL
LIN {X 0,Y 580.335,Z 262.509,A -85,B 0,C 180,E1 -1802.776,E2 -1802.776} C_VEL
LIN {X 0,Y 580.328,Z 262.505,A -85,B 0,C 180,E1 -1805.56,E2 -1805.56} C_VEL
LIN {X 0,Y 580.326,Z 262.505,A -85,B 0,C 180,E1 -1808.356,E2 -1808.356} C_VEL
LIN {X 0,Y 580.297,Z 262.512,A -85,B 0,C 180,E1 -1811.191,E2 -1811.191} C_VEL
LIN {X 0,Y 580.323,Z 262.504,A -85,B 0,C 180,E1 -1814.017,E2 -1814.017} C_VEL
LIN {X 0,Y 580.309,Z 262.516,A -85,B 0,C 180,E1 -1816.914,E2 -1816.914} C_VEL
LIN {X 0,Y 580.301,Z 262.507,A -85,B 0,C 180,E1 -1819.822,E2 -1819.822} C_VEL
LIN {X 0,Y 580.292,Z 262.517,A -85,B 0,C 180,E1 -1822.802,E2 -1822.802} C_VEL
LIN {X 0,Y 580.302,Z 262.514,A -85,B 0,C 180,E1 -1825.08,E2 -1825.08} C_VEL
LIN {X 0,Y 580.296,Z 262.509,A -85,B 0,C 180,E1 -1828.186,E2 -1828.186} C_VEL
LIN {X 0,Y 580.282,Z 262.518,A -85,B 0,C 180,E1 -1830.695,E2 -1830.695} C_VEL
LIN {X 0,Y 580.299,Z 262.511,A -85,B 0,C 180,E1 -1833.316,E2 -1833.316} C_VEL
LIN {X 0,Y 580.323,Z 262.504,A -85,B 0,C 180,E1 -1835.767,E2 -1835.767} C_VEL
LIN {X 0,Y 580.285,Z 262.511,A -85,B 0,C 180,E1 -1838.146,E2 -1838.146} C_VEL
LIN {X 0,Y 580.299,Z 262.517,A -85,B 0,C 180,E1 -1840.843,E2 -1840.843} C_VEL
LIN {X 0,Y 580.275,Z 262.511,A -85,B 0,C 180,E1 -1843.658,E2 -1843.658} C_VEL
LIN {X 0,Y 580.282,Z 262.518,A -85,B 0,C 180,E1 -1846.609,E2 -1846.609} C_VEL
LIN {X 0,Y 580.297,Z 262.512,A -85,B 0,C 180,E1 -1849.157,E2 -1849.157} C_VEL
LIN {X 0,Y 580.286,Z 262.51,A -85,B 0,C 180,E1 -1851.927,E2 -1851.927} C_VEL
LIN {X 0,Y 580.251,Z 262.52,A -85,B 0,C 180,E1 -1854.453,E2 -1854.453} C_VEL
LIN {X 0,Y 580.287,Z 262.515,A -85,B 0,C 180,E1 -1856.975,E2 -1856.975} C_VEL
LIN {X 0,Y 580.295,Z 262.51,A -85,B 0,C 180,E1 -1859.425,E2 -1859.425} C_VEL
LIN {X 0,Y 580.329,Z 262.612,A -85,B 0,C 180,E1 -1862.259,E2 -1862.259} C_VEL
LIN {X 0,Y 582.194,Z 269.676,A -85,B 0,C 180,E1 -1862.978,E2 -1862.978} C_VEL
LIN {X 0,Y 581.901,Z 297.412,A -85,B 0,C 180,E1 -1865.378,E2 -1865.378} C_VEL
LIN {X 0,Y 581.767,Z 311.895,A -85,B 0,C 180,E1 -1866.614,E2 -1866.614} C_VEL
LIN {X 0,Y 582.717,Z 318.174,A -85,B 0,C 180,E1 -1866.748,E2 -1866.748} C_VEL
LIN {X 0,Y 582.136,Z 519.44,A -85,B 0,C 180,E1 -1869.368,E2 -1869.368} C_VEL
LIN {X 0,Y 582.05,Z 536.011,A -85,B 0,C 180,E1 -1869.734,E2 -1869.734} C_VEL
LIN {X 0,Y 581.824,Z 552.246,A -85,B 0,C 180,E1 -1870.232,E2 -1870.232} C_VEL
LIN {X 0,Y 581.6,Z 569.053,A -85,B 0,C 180,E1 -1870.91,E2 -1870.91} C_VEL
LIN {X 0,Y 581.414,Z 584.306,A -85,B 0,C 180,E1 -1871.683,E2 -1871.683} C_VEL
LIN {X 0,Y 581.161,Z 598.785,A -85,B 0,C 180,E1 -1872.567,E2 -1872.567} C_VEL
LIN {X 0,Y 580.977,Z 612.543,A -85,B 0,C 180,E1 -1873.575,E2 -1873.575} C_VEL
LIN {X 0,Y 580.742,Z 624.074,A -85,B 0,C 180,E1 -1874.56,E2 -1874.56} C_VEL
LIN {X 0,Y 580.589,Z 635.622,A -85,B 0,C 180,E1 -1875.7,E2 -1875.7} C_VEL
LIN {X 0,Y 580.412,Z 647.335,A -85,B 0,C 180,E1 -1877.055,E2 -1877.055} C_VEL
LIN {X 0,Y 580.315,Z 657.677,A -85,B 0,C 180,E1 -1878.474,E2 -1878.474} C_VEL
LIN {X 0,Y 580.219,Z 666.286,A -85,B 0,C 180,E1 -1879.885,E2 -1879.885} C_VEL
LIN {X 0,Y 580.164,Z 673.488,A -85,B 0,C 180,E1 -1881.291,E2 -1881.291} C_VEL
LIN {X 0,Y 580.119,Z 679.467,A -85,B 0,C 180,E1 -1882.692,E2 -1882.692} C_VEL
LIN {X 0,Y 580.111,Z 685.247,A -85,B 0,C 180,E1 -1884.438,E2 -1884.438} C_VEL
LIN {X 0,Y 580.086,Z 688.635,A -85,B 0,C 180,E1 -1885.831,E2 -1885.831} C_VEL
LIN {X 0,Y 580.031,Z 691.088,A -85,B 0,C 180,E1 -1887.222,E2 -1887.222} C_VEL
LIN {X 0,Y 580.04,Z 692.479,A -85,B 0,C 180,E1 -1888.611,E2 -1888.611} C_VEL
LIN {X 0,Y 580.033,Z 693,A -85,B 0,C 180,E1 -1890,E2 -1890} C_VEL
LIN {X 0,Y 580.04,Z 692.479,A -85,B 0,C 180,E1 -1891.389,E2 -1891.389} C_VEL
LIN {X 0,Y 580.031,Z 691.088,A -85,B 0,C 180,E1 -1892.778,E2 -1892.778} C_VEL
LIN {X 0,Y 580.086,Z 688.635,A -85,B 0,C 180,E1 -1894.169,E2 -1894.169} C_VEL
LIN {X 0,Y 580.098,Z 684.187,A -85,B 0,C 180,E1 -1895.911,E2 -1895.911} C_VEL
LIN {X 0,Y 580.119,Z 679.468,A -85,B 0,C 180,E1 -1897.308,E2 -1897.308} C_VEL
LIN {X 0,Y 580.156,Z 671.857,A -85,B 0,C 180,E1 -1899.061,E2 -1899.061} C_VEL
LIN {X 0,Y 580.24,Z 663.25,A -85,B 0,C 180,E1 -1900.644,E2 -1900.644} C_VEL
LIN {X 0,Y 580.335,Z 653.973,A -85,B 0,C 180,E1 -1902.058,E2 -1902.058} C_VEL
LIN {X 0,Y 580.44,Z 644.425,A -85,B 0,C 180,E1 -1903.3,E2 -1903.3} C_VEL
LIN {X 0,Y 580.623,Z 632.932,A -85,B 0,C 180,E1 -1904.582,E2 -1904.582} C_VEL
LIN {X 0,Y 580.814,Z 621.144,A -85,B 0,C 180,E1 -1905.708,E2 -1905.708} C_VEL
LIN {X 0,Y 581.011,Z 607.878,A -85,B 0,C 180,E1 -1906.786,E2 -1906.786} C_VEL
LIN {X 0,Y 581.263,Z 593.432,A -85,B 0,C 180,E1 -1907.776,E2 -1907.776} C_VEL
LIN {X 0,Y 581.478,Z 579.274,A -85,B 0,C 180,E1 -1908.589,E2 -1908.589} C_VEL
LIN {X 0,Y 581.696,Z 564.012,A -85,B 0,C 180,E1 -1909.314,E2 -1909.314} C_VEL
LIN {X 0,Y 581.904,Z 548.348,A -85,B 0,C 180,E1 -1909.903,E2 -1909.903} C_VEL
LIN {X 0,Y 582.055,Z 532.356,A -85,B 0,C 180,E1 -1910.359,E2 -1910.359} C_VEL
LIN {X 0,Y 582.148,Z 516.442,A -85,B 0,C 180,E1 -1910.678,E2 -1910.678} C_VEL
LIN {X 0,Y 582.717,Z 317.363,A -85,B 0,C 180,E1 -1913.263,E2 -1913.263} C_VEL
LIN {X 0,Y 581.753,Z 311.95,A -85,B 0,C 180,E1 -1913.382,E2 -1913.382} C_VEL
LIN {X 0,Y 582.175,Z 277.509,A -85,B 0,C 180,E1 -1916.336,E2 -1916.336} C_VEL
LIN {X 0,Y 582.193,Z 269.672,A -85,B 0,C 180,E1 -1917.022,E2 -1917.022} C_VEL
LIN {X 0,Y 580.31,Z 262.513,A -85,B 0,C 180,E1 -1917.767,E2 -1917.767} C_VEL
LIN {X 0,Y 580.285,Z 262.512,A -85,B 0,C 180,E1 -1920.695,E2 -1920.695} C_VEL
LIN {X 0,Y 580.301,Z 262.515,A -85,B 0,C 180,E1 -1923.316,E2 -1923.316} C_VEL
LIN {X 0,Y 580.247,Z 262.517,A -85,B 0,C 180,E1 -1925.757,E2 -1925.757} C_VEL
LIN {X 0,Y 580.286,Z 262.51,A -85,B 0,C 180,E1 -1928.146,E2 -1928.146} C_VEL
LIN {X 0,Y 580.296,Z 262.511,A -85,B 0,C 180,E1 -1930.843,E2 -1930.843} C_VEL
LIN {X 0,Y 580.285,Z 262.513,A -85,B 0,C 180,E1 -1933.657,E2 -1933.657} C_VEL
LIN {X 0,Y 580.273,Z 262.511,A -85,B 0,C 180,E1 -1936.609,E2 -1936.609} C_VEL
LIN {X 0,Y 580.299,Z 262.515,A -85,B 0,C 180,E1 -1939.157,E2 -1939.157} C_VEL
LIN {X 0,Y 580.287,Z 262.509,A -85,B 0,C 180,E1 -1941.927,E2 -1941.927} C_VEL
LIN {X 0,Y 580.285,Z 262.509,A -85,B 0,C 180,E1 -1944.455,E2 -1944.455} C_VEL
LIN {X 0,Y 580.287,Z 262.515,A -85,B 0,C 180,E1 -1946.975,E2 -1946.975} C_VEL
LIN {X 0,Y 580.293,Z 262.514,A -85,B 0,C 180,E1 -1949.425,E2 -1949.425} C_VEL
LIN {X 0,Y 580.295,Z 262.507,A -85,B 0,C 180,E1 -1952.141,E2 -1952.141} C_VEL
LIN {X 0,Y 580.318,Z 262.513,A -85,B 0,C 180,E1 -1955.27,E2 -1955.27} C_VEL
LIN {X 0,Y 580.269,Z 262.511,A -85,B 0,C 180,E1 -1957.947,E2 -1957.947} C_VEL
LIN {X 0,Y 580.296,Z 262.511,A -85,B 0,C 180,E1 -1960.913,E2 -1960.913} C_VEL
LIN {X 0,Y 580.276,Z 262.511,A -85,B 0,C 180,E1 -1963.826,E2 -1963.826} C_VEL
LIN {X 0,Y 580.323,Z 262.501,A -85,B 0,C 180,E1 -1965.983,E2 -1965.983} C_VEL
LIN {X 0,Y 580.302,Z 262.511,A -85,B 0,C 180,E1 -1968.827,E2 -1968.827} C_VEL
LIN {X 0,Y 580.326,Z 262.504,A -85,B 0,C 180,E1 -1971.644,E2 -1971.644} C_VEL
LIN {X 0,Y 580.327,Z 262.502,A -85,B 0,C 180,E1 -1974.44,E2 -1974.44} C_VEL
LIN {X 0,Y 580.336,Z 262.51,A -85,B 0,C 180,E1 -1977.224,E2 -1977.224} C_VEL
LIN {X 0,Y 580.351,Z 262.498,A -85,B 0,C 180,E1 -1980,E2 -1980} C_VEL
LIN {X 0,Y 580.335,Z 262.507,A -85,B 0,C 180,E1 -1982.777,E2 -1982.777} C_VEL
LIN {X 0,Y 580.328,Z 262.505,A -85,B 0,C 180,E1 -1985.56,E2 -1985.56} C_VEL
LIN {X 0,Y 580.326,Z 262.501,A -85,B 0,C 180,E1 -1988.356,E2 -1988.356} C_VEL
LIN {X 0,Y 580.298,Z 262.514,A -85,B 0,C 180,E1 -1991.191,E2 -1991.191} C_VEL
LIN {X 0,Y 580.324,Z 262.502,A -85,B 0,C 180,E1 -1994.017,E2 -1994.017} C_VEL
LIN {X 0,Y 580.31,Z 262.513,A -85,B 0,C 180,E1 -1996.914,E2 -1996.914} C_VEL
LIN {X 0,Y 580.302,Z 262.506,A -85,B 0,C 180,E1 -1999.822,E2 -1999.822} C_VEL
LIN {X 0,Y 580.281,Z 262.51,A -85,B 0,C 180,E1 -2001.326,E2 -2001.326} C_VEL
LIN {X 0,Y 579.584,Z 262.595,A -85,B 0,C 180,E1 -2001.906,E2 -2001.906} C_VEL
LIN {X 0,Y 576.708,Z 262.96,A -85,B 0,C 180,E1 -2002.846,E2 -2002.846} C_VEL
LIN {X 0,Y 574.314,Z 263.255,A -85,B 0,C 180,E1 -2003.602,E2 -2003.602} C_VEL
LIN {X 0,Y 573.315,Z 263.378,A -85,B 0,C 180,E1 -2004.186,E2 -2004.186} C_VEL
LIN {X 0,Y 573.248,Z 263.387,A -85,B 0,C 180,E1 -2004.383,E2 -2004.383} C_VEL
LIN {X 0,Y 573.248,Z 263.391,A -85,B 0,C 180,E1 -2006.976,E2 -2006.976} C_VEL
LIN {X 0,Y 573.245,Z 263.388,A -85,B 0,C 180,E1 -2009.489,E2 -2009.489} C_VEL
LIN {X 0,Y 573.251,Z 263.391,A -85,B 0,C 180,E1 -2012.645,E2 -2012.645} C_VEL
LIN {X 0,Y 573.267,Z 263.388,A -85,B 0,C 180,E1 -2015.184,E2 -2015.184} C_VEL
LIN {X 0,Y 573.235,Z 263.385,A -85,B 0,C 180,E1 -2017.808,E2 -2017.808} C_VEL
LIN {X 0,Y 573.243,Z 263.391,A -85,B 0,C 180,E1 -2020.525,E2 -2020.525} C_VEL
LIN {X 0,Y 573.238,Z 263.389,A -85,B 0,C 180,E1 -2023.359,E2 -2023.359} C_VEL
LIN {X 0,Y 573.251,Z 263.386,A -85,B 0,C 180,E1 -2026.33,E2 -2026.33} C_VEL
LIN {X 0,Y 573.258,Z 263.386,A -85,B 0,C 180,E1 -2029.476,E2 -2029.476} C_VEL
LIN {X 0,Y 573.235,Z 263.388,A -85,B 0,C 180,E1 -2032.193,E2 -2032.193} C_VEL
LIN {X 0,Y 573.233,Z 263.391,A -85,B 0,C 180,E1 -2035.229,E2 -2035.229} C_VEL
LIN {X 0,Y 573.25,Z 263.386,A -85,B 0,C 180,E1 -2037.772,E2 -2037.772} C_VEL
LIN {X 0,Y 573.26,Z 263.393,A -85,B 0,C 180,E1 -2040.634,E2 -2040.634} C_VEL
LIN {X 0,Y 573.25,Z 263.394,A -85,B 0,C 180,E1 -2043.024,E2 -2043.024} C_VEL
LIN {X 0,Y 573.282,Z 263.582,A -85,B 0,C 180,E1 -2044.397,E2 -2044.397} C_VEL
LIN {X 0,Y 574.998,Z 270.83,A -85,B 0,C 180,E1 -2045.2,E2 -2045.2} C_VEL
LIN {X 0,Y 574.812,Z 282.831,A -85,B 0,C 180,E1 -2046.377,E2 -2046.377} C_VEL
LIN {X 0,Y 576.196,Z 290.017,A -85,B 0,C 180,E1 -2046.538,E2 -2046.538} C_VEL
LIN {X 0,Y 575.497,Z 488.063,A -85,B 0,C 180,E1 -2049.142,E2 -2049.142} C_VEL
LIN {X 0,Y 575.371,Z 504.254,A -85,B 0,C 180,E1 -2049.488,E2 -2049.488} C_VEL
LIN {X 0,Y 575.136,Z 520.989,A -85,B 0,C 180,E1 -2049.992,E2 -2049.992} C_VEL
LIN {X 0,Y 574.917,Z 537.181,A -85,B 0,C 180,E1 -2050.637,E2 -2050.637} C_VEL
LIN {X 0,Y 574.666,Z 551.92,A -85,B 0,C 180,E1 -2051.367,E2 -2051.367} C_VEL
LIN {X 0,Y 574.38,Z 566.822,A -85,B 0,C 180,E1 -2052.269,E2 -2052.269} C_VEL
LIN {X 0,Y 574.107,Z 580.813,A -85,B 0,C 180,E1 -2053.281,E2 -2053.281} C_VEL
LIN {X 0,Y 573.846,Z 593.589,A -85,B 0,C 180,E1 -2054.369,E2 -2054.369} C_VEL
LIN {X 0,Y 573.632,Z 605.86,A -85,B 0,C 180,E1 -2055.594,E2 -2055.594} C_VEL
LIN {X 0,Y 573.419,Z 616.997,A -85,B 0,C 180,E1 -2056.895,E2 -2056.895} C_VEL
LIN {X 0,Y 573.287,Z 627.366,A -85,B 0,C 180,E1 -2058.33,E2 -2058.33} C_VEL
LIN {X 0,Y 573.176,Z 636.031,A -85,B 0,C 180,E1 -2059.759,E2 -2059.759} C_VEL
LIN {X 0,Y 573.084,Z 643.284,A -85,B 0,C 180,E1 -2061.182,E2 -2061.182} C_VEL
LIN {X 0,Y 573.042,Z 649.292,A -85,B 0,C 180,E1 -2062.601,E2 -2062.601} C_VEL
LIN {X 0,Y 573.014,Z 654.052,A -85,B 0,C 180,E1 -2064.016,E2 -2064.016} C_VEL
LIN {X 0,Y 573.008,Z 658.544,A -85,B 0,C 180,E1 -2065.78,E2 -2065.78} C_VEL
LIN {X 0,Y 572.948,Z 661.019,A -85,B 0,C 180,E1 -2067.188,E2 -2067.188} C_VEL
LIN {X 0,Y 572.941,Z 662.449,A -85,B 0,C 180,E1 -2068.594,E2 -2068.594} C_VEL
LIN {X 0,Y 572.935,Z 662.996,A -85,B 0,C 180,E1 -2070,E2 -2070} C_VEL
LIN {X 0,Y 572.938,Z 662.509,A -85,B 0,C 180,E1 -2071.406,E2 -2071.406} C_VEL
LIN {X 0,Y 572.948,Z 661.15,A -85,B 0,C 180,E1 -2072.812,E2 -2072.812} C_VEL
LIN {X 0,Y 573.005,Z 658.728,A -85,B 0,C 180,E1 -2074.22,E2 -2074.22} C_VEL
LIN {X 0,Y 573.038,Z 655.379,A -85,B 0,C 180,E1 -2075.631,E2 -2075.631} C_VEL
LIN {X 0,Y 573.045,Z 650.875,A -85,B 0,C 180,E1 -2077.045,E2 -2077.045} C_VEL
LIN {X 0,Y 573.083,Z 645.307,A -85,B 0,C 180,E1 -2078.462,E2 -2078.462} C_VEL
LIN {X 0,Y 573.14,Z 638.463,A -85,B 0,C 180,E1 -2079.885,E2 -2079.885} C_VEL
LIN {X 0,Y 573.251,Z 630.216,A -85,B 0,C 180,E1 -2081.312,E2 -2081.312} C_VEL
LIN {X 0,Y 573.393,Z 620.395,A -85,B 0,C 180,E1 -2082.746,E2 -2082.746} C_VEL
LIN {X 0,Y 573.567,Z 610.294,A -85,B 0,C 180,E1 -2084.004,E2 -2084.004} C_VEL
LIN {X 0,Y 573.738,Z 598.387,A -85,B 0,C 180,E1 -2085.27,E2 -2085.27} C_VEL
LIN {X 0,Y 574.016,Z 585.306,A -85,B 0,C 180,E1 -2086.447,E2 -2086.447} C_VEL
LIN {X 0,Y 574.284,Z 572.168,A -85,B 0,C 180,E1 -2087.453,E2 -2087.453} C_VEL
LIN {X 0,Y 574.534,Z 558.224,A -85,B 0,C 180,E1 -2088.36,E2 -2088.36} C_VEL
LIN {X 0,Y 574.799,Z 543.015,A -85,B 0,C 180,E1 -2089.183,E2 -2089.183} C_VEL
LIN {X 0,Y 575.09,Z 526.459,A -85,B 0,C 180,E1 -2089.901,E2 -2089.901} C_VEL
LIN {X 0,Y 575.313,Z 510.117,A -85,B 0,C 180,E1 -2090.444,E2 -2090.444} C_VEL
LIN {X 0,Y 575.457,Z 493.982,A -85,B 0,C 180,E1 -2090.836,E2 -2090.836} C_VEL
LIN {X 0,Y 575.596,Z 474.874,A -85,B 0,C 180,E1 -2091.135,E2 -2091.135} C_VEL
LIN {X 0,Y 576.171,Z 289.621,A -85,B 0,C 180,E1 -2093.558,E2 -2093.558} C_VEL
LIN {X 0,Y 574.787,Z 282.755,A -85,B 0,C 180,E1 -2093.722,E2 -2093.722} C_VEL
LIN {X 0,Y 574.927,Z 270.24,A -85,B 0,C 180,E1 -2094.952,E2 -2094.952} C_VEL
LIN {X 0,Y 573.262,Z 263.392,A -85,B 0,C 180,E1 -2095.726,E2 -2095.726} C_VEL
LIN {X 0,Y 573.23,Z 263.391,A -85,B 0,C 180,E1 -2098.565,E2 -2098.565} C_VEL
LIN {X 0,Y 573.224,Z 263.395,A -85,B 0,C 180,E1 -2100.993,E2 -2100.993} C_VEL
LIN {X 0,Y 573.262,Z 263.392,A -85,B 0,C 180,E1 -2103.524,E2 -2103.524} C_VEL
LIN {X 0,Y 573.192,Z 263.391,A -85,B 0,C 180,E1 -2106.053,E2 -2106.053} C_VEL
LIN {X 0,Y 573.238,Z 263.389,A -85,B 0,C 180,E1 -2108.702,E2 -2108.702} C_VEL
LIN {X 0,Y 573.236,Z 263.391,A -85,B 0,C 180,E1 -2111.593,E2 -2111.593} C_VEL
LIN {X 0,Y 573.238,Z 263.387,A -85,B 0,C 180,E1 -2114.333,E2 -2114.333} C_VEL
LIN {X 0,Y 573.238,Z 263.395,A -85,B 0,C 180,E1 -2117.358,E2 -2117.358} C_VEL
LIN {X 0,Y 573.238,Z 263.387,A -85,B 0,C 180,E1 -2120.392,E2 -2120.392} C_VEL
LIN {X 0,Y 573.253,Z 263.392,A -85,B 0,C 180,E1 -2123.078,E2 -2123.078} C_VEL
LIN {X 0,Y 573.268,Z 263.385,A -85,B 0,C 180,E1 -2125.671,E2 -2125.671} C_VEL
LIN {X 0,Y 573.238,Z 263.386,A -85,B 0,C 180,E1 -2128.184,E2 -2128.184} C_VEL
LIN {X 0,Y 573.262,Z 263.386,A -85,B 0,C 180,E1 -2130.634,E2 -2130.634} C_VEL
LIN {X 0,Y 573.248,Z 263.391,A -85,B 0,C 180,E1 -2133.024,E2 -2133.024} C_VEL
LIN {X 0,Y 573.273,Z 263.388,A -85,B 0,C 180,E1 -2135.366,E2 -2135.366} C_VEL
LIN {X 0,Y 573.226,Z 263.386,A -85,B 0,C 180,E1 -2138.419,E2 -2138.419} C_VEL
LIN {X 0,Y 573.266,Z 263.387,A -85,B 0,C 180,E1 -2140.731,E2 -2140.731} C_VEL
LIN {X 0,Y 573.248,Z 263.384,A -85,B 0,C 180,E1 -2143.622,E2 -2143.622} C_VEL
LIN {X 0,Y 573.271,Z 263.383,A -85,B 0,C 180,E1 -2145.807,E2 -2145.807} C_VEL
LIN {X 0,Y 573.26,Z 263.389,A -85,B 0,C 180,E1 -2148.745,E2 -2148.745} C_VEL
LIN {X 0,Y 573.282,Z 263.383,A -85,B 0,C 180,E1 -2151.54,E2 -2151.54} C_VEL
LIN {X 0,Y 573.296,Z 263.381,A -85,B 0,C 180,E1 -2154.372,E2 -2154.372} C_VEL
LIN {X 0,Y 573.312,Z 263.375,A -85,B 0,C 180,E1 -2157.892,E2 -2157.892} C_VEL
LIN {X 0,Y 573.329,Z 263.381,A -85,B 0,C 180,E1 -2160.702,E2 -2160.702} C_VEL
LIN {X 0,Y 573.302,Z 263.385,A -85,B 0,C 180,E1 -2162.811,E2 -2162.811} C_VEL
LIN {X 0,Y 573.296,Z 263.38,A -85,B 0,C 180,E1 -2165.628,E2 -2165.628} C_VEL
LIN {X 0,Y 573.281,Z 263.384,A -85,B 0,C 180,E1 -2168.459,E2 -2168.459} C_VEL
LIN {X 0,Y 573.269,Z 263.386,A -85,B 0,C 180,E1 -2171.312,E2 -2171.312} C_VEL
LIN {X 0,Y 573.278,Z 263.385,A -85,B 0,C 180,E1 -2174.425,E2 -2174.425} C_VEL
LIN {X 0,Y 573.255,Z 263.391,A -85,B 0,C 180,E1 -2177.112,E2 -2177.112} C_VEL
LIN {X 0,Y 573.249,Z 263.386,A -85,B 0,C 180,E1 -2180.077,E2 -2180.077} C_VEL
LIN {X 0,Y 573.231,Z 263.394,A -85,B 0,C 180,E1 -2183.099,E2 -2183.099} C_VEL
LIN {X 0,Y 573.249,Z 263.388,A -85,B 0,C 180,E1 -2185.41,E2 -2185.41} C_VEL
LIN {X 0,Y 573.248,Z 263.386,A -85,B 0,C 180,E1 -2188.029,E2 -2188.029} C_VEL
LIN {X 0,Y 573.243,Z 263.388,A -85,B 0,C 180,E1 -2190.176,E2 -2190.176} C_VEL
LIN {X 0,Y 573.25,Z 263.394,A -85,B 0,C 180,E1 -2192.645,E2 -2192.645} C_VEL
LIN {X 0,Y 573.266,Z 263.388,A -85,B 0,C 180,E1 -2195.184,E2 -2195.184} C_VEL
LIN {X 0,Y 573.233,Z 263.388,A -85,B 0,C 180,E1 -2197.808,E2 -2197.808} C_VEL
LIN {X 0,Y 573.267,Z 263.39,A -85,B 0,C 180,E1 -2200.528,E2 -2200.528} C_VEL
LIN {X 0,Y 573.241,Z 263.387,A -85,B 0,C 180,E1 -2203.669,E2 -2203.669} C_VEL
LIN {X 0,Y 573.243,Z 263.396,A -85,B 0,C 180,E1 -2206.642,E2 -2206.642} C_VEL
LIN {X 0,Y 573.256,Z 263.386,A -85,B 0,C 180,E1 -2209.476,E2 -2209.476} C_VEL
LIN {X 0,Y 573.232,Z 263.391,A -85,B 0,C 180,E1 -2212.193,E2 -2212.193} C_VEL
LIN {X 0,Y 573.232,Z 263.388,A -85,B 0,C 180,E1 -2215.229,E2 -2215.229} C_VEL
LIN {X 0,Y 573.248,Z 263.387,A -85,B 0,C 180,E1 -2217.772,E2 -2217.772} C_VEL
LIN {X 0,Y 573.258,Z 263.394,A -85,B 0,C 180,E1 -2220.634,E2 -2220.634} C_VEL
LIN {X 0,Y 573.249,Z 263.398,A -85,B 0,C 180,E1 -2221.971,E2 -2221.971} C_VEL
LIN {X 0,Y 575.527,Z 271.311,A -85,B 0,C 180,E1 -2222.786,E2 -2222.786} C_VEL
LIN {X 0,Y 575.306,Z 292.968,A -85,B 0,C 180,E1 -2224.687,E2 -2224.687} C_VEL
LIN {X 0,Y 575.029,Z 311.959,A -85,B 0,C 180,E1 -2226.329,E2 -2226.329} C_VEL
LIN {X 0,Y 576.224,Z 319.199,A -85,B 0,C 180,E1 -2226.484,E2 -2226.484} C_VEL
LIN {X 0,Y 575.509,Z 517.949,A -85,B 0,C 180,E1 -2229.096,E2 -2229.096} C_VEL
LIN {X 0,Y 575.354,Z 534.185,A -85,B 0,C 180,E1 -2229.441,E2 -2229.441} C_VEL
LIN {X 0,Y 575.117,Z 550.947,A -85,B 0,C 180,E1 -2229.945,E2 -2229.945} C_VEL
LIN {X 0,Y 574.932,Z 566.282,A -85,B 0,C 180,E1 -2230.55,E2 -2230.55} C_VEL
LIN {X 0,Y 574.665,Z 581.03,A -85,B 0,C 180,E1 -2231.275,E2 -2231.275} C_VEL
LIN {X 0,Y 574.432,Z 594.857,A -85,B 0,C 180,E1 -2232.098,E2 -2232.098} C_VEL
LIN {X 0,Y 574.13,Z 609.05,A -85,B 0,C 180,E1 -2233.099,E2 -2233.099} C_VEL
LIN {X 0,Y 573.88,Z 622.122,A -85,B 0,C 180,E1 -2234.188,E2 -2234.188} C_VEL
LIN {X 0,Y 573.658,Z 633.983,A -85,B 0,C 180,E1 -2235.344,E2 -2235.344} C_VEL
LIN {X 0,Y 573.448,Z 645.909,A -85,B 0,C 180,E1 -2236.715,E2 -2236.715} C_VEL
LIN {X 0,Y 573.269,Z 656.444,A -85,B 0,C 180,E1 -2238.15,E2 -2238.15} C_VEL
LIN {X 0,Y 573.181,Z 665.276,A -85,B 0,C 180,E1 -2239.581,E2 -2239.581} C_VEL
LIN {X 0,Y 573.077,Z 673.489,A -85,B 0,C 180,E1 -2241.182,E2 -2241.182} C_VEL
LIN {X 0,Y 573.04,Z 679.467,A -85,B 0,C 180,E1 -2242.601,E2 -2242.601} C_VEL
LIN {X 0,Y 573.014,Z 684.186,A -85,B 0,C 180,E1 -2244.016,E2 -2244.016} C_VEL
LIN {X 0,Y 573.006,Z 688.636,A -85,B 0,C 180,E1 -2245.78,E2 -2245.78} C_VEL
LIN {X 0,Y 572.947,Z 691.089,A -85,B 0,C 180,E1 -2247.188,E2 -2247.188} C_VEL
LIN {X 0,Y 572.939,Z 692.479,A -85,B 0,C 180,E1 -2248.594,E2 -2248.594} C_VEL
LIN {X 0,Y 572.933,Z 693,A -85,B 0,C 180,E1 -2250,E2 -2250} C_VEL
LIN {X 0,Y 572.939,Z 692.479,A -85,B 0,C 180,E1 -2251.406,E2 -2251.406} C_VEL
LIN {X 0,Y 572.947,Z 691.088,A -85,B 0,C 180,E1 -2252.812,E2 -2252.812} C_VEL
LIN {X 0,Y 573.006,Z 688.635,A -85,B 0,C 180,E1 -2254.22,E2 -2254.22} C_VEL
LIN {X 0,Y 573.013,Z 684.188,A -85,B 0,C 180,E1 -2255.984,E2 -2255.984} C_VEL
LIN {X 0,Y 573.04,Z 679.468,A -85,B 0,C 180,E1 -2257.399,E2 -2257.399} C_VEL
LIN {X 0,Y 573.076,Z 673.489,A -85,B 0,C 180,E1 -2258.818,E2 -2258.818} C_VEL
LIN {X 0,Y 573.182,Z 665.276,A -85,B 0,C 180,E1 -2260.42,E2 -2260.42} C_VEL
LIN {X 0,Y 573.269,Z 656.445,A -85,B 0,C 180,E1 -2261.85,E2 -2261.85} C_VEL
LIN {X 0,Y 573.448,Z 645.909,A -85,B 0,C 180,E1 -2263.285,E2 -2263.285} C_VEL
LIN {X 0,Y 573.59,Z 635.035,A -85,B 0,C 180,E1 -2264.544,E2 -2264.544} C_VEL
LIN {X 0,Y 573.831,Z 624.071,A -85,B 0,C 180,E1 -2265.631,E2 -2265.631} C_VEL
LIN {X 0,Y 574.091,Z 610.222,A -85,B 0,C 180,E1 -2266.811,E2 -2266.811} C_VEL
